C08947=1013.644,84.110,-119.825,166.038,58.565,160.621
C08948=1013.639,83.861,-119.809,166.035,58.575,160.623
C08949=1013.634,83.612,-119.793,166.034,58.586,160.624
C08950=1013.630,83.362,-119.778,166.031,58.596,160.626
C08951=1013.625,83.112,-119.762,166.029,58.606,160.627
C08952=1013.621,82.863,-119.746,166.027,58.617,160.629
C08953=1013.617,82.613,-119.730,166.025,58.627,160.630
C08954=1013.612,82.364,-119.715,166.022,58.638,160.632
C08955=1013.608,82.114,-119.699,166.021,58.647,160.633
C08956=1013.604,81.864,-119.683,166.018,58.658,160.634
C08957=1013.599,81.615,-119.668,166.016,58.669,160.636
C08958=1013.595,81.366,-119.652,166.014,58.678,160.637
C08959=1013.590,81.116,-119.636,166.011,58.689,160.639
C08960=1013.586,80.866,-119.621,166.009,58.699,160.640
C08961=1013.582,80.617,-119.605,166.007,58.709,160.642
C08962=1013.577,80.367,-119.589,166.004,58.719,160.643
C08963=1013.574,80.118,-119.574,166.002,58.730,160.644
C08964=1013.569,79.869,-119.558,166.000,58.740,160.646
C08965=1013.564,79.620,-119.543,165.997,58.750,160.647
C08966=1013.560,79.370,-119.527,165.996,58.760,160.649
C08967=1013.556,79.120,-119.511,165.994,58.771,160.650
C08968=1013.551,78.871,-119.495,165.992,58.781,160.652
C08969=1013.547,78.621,-119.480,165.989,58.791,160.653
C08970=1013.543,78.372,-119.464,165.986,58.801,160.654
C08971=1013.538,78.122,-119.448,165.984,58.811,160.656
C08972=1013.534,77.873,-119.432,165.982,58.822,160.657
C08973=1013.530,77.624,-119.417,165.981,58.832,160.659
C08974=1013.525,77.374,-119.402,165.978,58.842,160.660
C08975=1013.521,77.125,-119.386,165.976,58.852,160.662
C08976=1013.517,76.875,-119.370,165.973,58.862,160.663
C08977=1013.512,76.626,-119.354,165.972,58.872,160.664
C08978=1013.508,76.375,-119.339,165.969,58.882,160.666
C08979=1013.503,76.126,-119.324,165.968,58.893,160.668
C08980=1013.499,75.877,-119.308,165.965,58.903,160.669
C08981=1013.495,75.628,-119.293,165.963,58.913,160.670
C08982=1013.490,75.378,-119.278,165.960,58.923,160.672
C08983=1013.486,75.128,-119.263,165.958,58.933,160.673
C08984=1013.482,74.879,-119.247,165.956,58.943,160.674
C08985=1013.476,74.600,-119.230,165.953,58.955,160.676
C08986=1013.471,74.320,-119.213,165.951,58.966,160.678
C08987=1013.467,74.040,-119.196,165.949,58.977,160.679
C08988=1013.462,73.761,-119.178,165.946,58.988,160.681
C08989=1013.457,73.511,-119.164,165.944,58.998,160.682
C08990=1013.453,73.261,-119.148,165.942,59.008,160.683
C08991=1013.448,73.013,-119.133,165.940,59.018,160.685
C08992=1013.444,72.763,-119.118,165.938,59.029,160.687
C08993=1013.440,72.513,-119.102,165.936,59.039,160.688
C08994=1013.435,72.264,-119.087,165.933,59.049,160.689
C08995=1013.431,72.014,-119.072,165.932,59.059,160.691
C08996=1013.427,71.765,-119.057,165.929,59.069,160.692
C08997=1013.422,71.515,-119.041,165.927,59.079,160.694
C08998=1013.417,71.266,-119.026,165.925,59.089,160.695
C08999=1013.413,71.016,-119.011,165.922,59.098,160.696
C09000=1013.409,70.766,-118.995,165.921,59.108,160.698
C09001=1013.404,70.518,-118.981,165.918,59.119,160.699
C09002=1013.400,70.268,-118.966,165.916,59.128,160.700
C09003=1013.395,70.018,-118.950,165.914,59.139,160.702
C09004=1013.391,69.768,-118.935,165.912,59.148,160.703
C09005=1013.387,69.520,-118.921,165.910,59.158,160.705
C09006=1013.383,69.270,-118.905,165.908,59.169,160.706
C09007=1013.378,69.020,-118.890,165.906,59.178,160.708
C09008=1013.374,68.771,-118.875,165.904,59.188,160.709
C09009=1013.370,68.520,-118.860,165.901,59.198,160.710
C09010=1013.365,68.272,-118.845,165.899,59.208,160.712
C09011=1013.361,68.022,-118.829,165.898,59.217,160.713
C09012=1013.356,67.772,-118.814,165.895,59.228,160.714
C09013=1013.352,67.523,-118.799,165.893,59.237,160.716
C09014=1013.348,67.274,-118.785,165.892,59.247,160.717
C09015=1013.343,67.024,-118.769,165.888,59.257,160.718
C09016=1013.339,66.774,-118.754,165.887,59.267,160.720
C09017=1013.334,66.525,-118.739,165.885,59.277,160.721
C09018=1013.330,66.276,-118.725,165.883,59.287,160.723
C09019=1013.325,66.026,-118.709,165.881,59.297,160.724
C09020=1013.320,65.776,-118.695,165.879,59.306,160.725
C09021=1013.317,65.527,-118.679,165.876,59.316,160.727
C09022=1013.312,65.277,-118.665,165.874,59.326,160.728
C09023=1013.307,65.027,-118.651,165.873,59.336,160.730
C09024=1013.303,64.778,-118.635,165.871,59.345,160.731
C09025=1013.299,64.529,-118.621,165.868,59.355,160.732
C09026=1013.294,64.279,-118.606,165.866,59.365,160.734
C09027=1013.290,64.029,-118.590,165.864,59.374,160.735
C09028=1013.286,63.780,-118.576,165.863,59.384,160.737
C09029=1013.281,63.531,-118.561,165.860,59.394,160.738
C09030=1013.277,63.281,-118.546,165.858,59.403,160.739
C09031=1013.272,63.032,-118.531,165.856,59.413,160.741
C09032=1013.267,62.782,-118.517,165.855,59.423,160.742
C09033=1013.263,62.532,-118.502,165.851,59.433,160.743
C09034=1013.259,62.283,-118.487,165.850,59.442,160.745
C09035=1013.254,62.034,-118.473,165.848,59.452,160.746
C09036=1013.250,61.784,-118.458,165.846,59.461,160.747
C09037=1013.245,61.534,-118.444,165.843,59.472,160.749
C09038=1013.241,61.285,-118.430,165.842,59.482,160.750
C09039=1013.236,61.035,-118.414,165.840,59.491,160.751
C09040=1013.231,60.786,-118.400,165.838,59.501,160.753
C09041=1013.227,60.536,-118.386,165.835,59.511,160.754
C09042=1013.222,60.286,-118.371,165.833,59.520,160.756
C09043=1013.218,60.037,-118.357,165.832,59.530,160.757
C09044=1013.213,59.787,-118.343,165.829,59.539,160.758
C09045=1013.208,59.537,-118.328,165.827,59.549,160.760
C09046=1013.204,59.289,-118.314,165.825,59.559,160.761
C09047=1013.199,59.039,-118.299,165.823,59.568,160.762
C09048=1013.195,58.790,-118.285,165.822,59.578,160.764
C09049=1013.190,58.510,-118.269,165.819,59.589,160.765
C09050=1013.185,58.230,-118.253,165.817,59.600,160.767
C09051=1013.180,57.951,-118.236,165.814,59.610,160.768
C09052=1013.175,57.671,-118.220,165.813,59.621,160.770
C09053=1013.170,57.421,-118.205,165.810,59.630,160.771
C09054=1013.166,57.172,-118.191,165.809,59.640,160.773
C09055=1013.161,56.922,-118.177,165.807,59.649,160.774
C09056=1013.157,56.673,-118.163,165.803,59.659,160.775
C09057=1013.152,56.423,-118.148,165.802,59.669,160.776
C09058=1013.148,56.173,-118.134,165.800,59.678,160.778
C09059=1013.144,55.924,-118.120,165.798,59.688,160.779
C09060=1013.139,55.674,-118.105,165.796,59.697,160.780
C09061=1013.134,55.426,-118.090,165.794,59.706,160.782
C09062=1013.130,55.176,-118.076,165.792,59.715,160.783
C09063=1013.126,54.927,-118.062,165.790,59.725,160.784
C09064=1013.121,54.677,-118.047,165.788,59.734,160.786
C09065=1013.117,54.428,-118.033,165.786,59.743,160.787
C09066=1013.112,54.178,-118.019,165.785,59.753,160.788
C09067=1013.107,53.928,-118.004,165.782,59.762,160.790
C09068=1013.103,53.679,-117.990,165.780,59.772,160.791
C09069=1013.098,53.429,-117.976,165.778,59.781,160.792
C09070=1013.094,53.180,-117.962,165.776,59.790,160.793
C09071=1013.089,52.930,-117.947,165.775,59.800,160.795
C09072=1013.085,52.681,-117.933,165.773,59.809,160.796
C09073=1013.081,52.431,-117.919,165.771,59.818,160.797
C09074=1013.076,52.181,-117.905,165.769,59.827,160.799
C09075=1013.072,51.932,-117.890,165.767,59.836,160.800
C09076=1013.068,51.682,-117.876,165.765,59.845,160.801
C09077=1013.063,51.432,-117.862,165.763,59.854,160.802
C09078=1013.059,51.183,-117.848,165.761,59.864,160.804
C09079=1013.054,50.933,-117.833,165.759,59.873,160.805
C09080=1013.050,50.684,-117.819,165.758,59.881,160.806
C09081=1013.045,50.434,-117.805,165.755,59.891,160.807
C09082=1013.041,50.185,-117.791,165.753,59.900,160.809
C09083=1013.036,49.935,-117.776,165.751,59.909,160.810
C09084=1013.032,49.686,-117.762,165.749,59.918,160.811
C09085=1013.027,49.436,-117.747,165.748,59.927,160.813
C09086=1013.023,49.187,-117.733,165.746,59.936,160.814
C09087=1013.018,48.937,-117.719,165.744,59.945,160.815
C09088=1013.014,48.688,-117.705,165.742,59.954,160.816
C09089=1013.010,48.438,-117.690,165.741,59.963,160.818
C09090=1013.005,48.189,-117.676,165.739,59.972,160.819
C09091=1013.001,47.938,-117.663,165.736,59.981,160.820
C09092=1012.997,47.689,-117.648,165.734,59.990,160.821
C09093=1012.992,47.439,-117.634,165.733,59.999,160.823
C09094=1012.988,47.190,-117.620,165.731,60.008,160.824
C09095=1012.983,46.940,-117.605,165.729,60.017,160.825
C09096=1012.979,46.691,-117.591,165.727,60.025,160.826
C09097=1012.975,46.442,-117.577,165.725,60.034,160.827
C09098=1012.970,46.192,-117.563,165.723,60.043,160.829
C09099=1012.966,45.943,-117.549,165.721,60.051,160.830
C09100=1012.961,45.693,-117.534,165.719,60.061,160.831
C09101=1012.957,45.444,-117.520,165.718,60.069,160.832
C09102=1012.953,45.193,-117.506,165.715,60.078,160.833
C09103=1012.949,44.944,-117.492,165.713,60.087,160.835
C09104=1012.944,44.695,-117.478,165.712,60.096,160.836
C09105=1012.940,44.445,-117.464,165.709,60.104,160.837
C09106=1012.936,44.196,-117.450,165.708,60.113,160.838
C09107=1012.931,43.946,-117.435,165.706,60.121,160.839
C09108=1012.927,43.697,-117.421,165.705,60.130,160.841
C09109=1012.923,43.448,-117.407,165.703,60.139,160.842
C09110=1012.918,43.197,-117.393,165.701,60.147,160.843
C09111=1012.914,42.948,-117.379,165.699,60.157,160.844
C09112=1012.909,42.698,-117.365,165.697,60.165,160.845
C09113=1012.903,42.319,-117.343,165.694,60.177,160.847
C09114=1012.896,41.941,-117.322,165.691,60.191,160.849
C09115=1012.890,41.563,-117.301,165.688,60.204,160.851
C09116=1012.883,41.184,-117.280,165.685,60.217,160.852
C09117=1012.878,40.936,-117.266,165.684,60.225,160.854
C09118=1012.874,40.685,-117.253,165.681,60.234,160.855
C09119=1012.870,40.436,-117.239,165.680,60.243,160.856
C09120=1012.866,40.187,-117.225,165.678,60.251,160.857
C09121=1012.860,39.936,-117.211,165.677,60.260,160.859
C09122=1012.856,39.687,-117.197,165.674,60.268,160.859
C09123=1012.852,39.437,-117.184,165.673,60.277,160.861
C09124=1012.847,39.188,-117.170,165.670,60.286,160.862
C09125=1012.843,38.939,-117.156,165.669,60.294,160.863
C09126=1012.838,38.688,-117.142,165.668,60.302,160.864
C09127=1012.834,38.439,-117.128,165.665,60.311,160.865
C09128=1012.830,38.190,-117.115,165.663,60.319,160.866
C09129=1012.825,37.940,-117.101,165.661,60.328,160.868
C09130=1012.821,37.690,-117.087,165.660,60.336,160.869
C09131=1012.816,37.441,-117.074,165.658,60.344,160.870
C09132=1012.812,37.191,-117.060,165.656,60.353,160.871
C09133=1012.808,36.941,-117.046,165.655,60.361,160.872
C09134=1012.803,36.692,-117.033,165.653,60.369,160.873
C09135=1012.799,36.443,-117.019,165.650,60.378,160.874
C09136=1012.794,36.193,-117.005,165.649,60.386,160.875
C09137=1012.777,48.138,-118.086,165.708,60.195,160.855
C09138=1012.781,48.387,-118.101,165.711,60.187,160.854
C09139=1012.785,48.637,-118.115,165.711,60.178,160.853
C09140=1012.790,48.886,-118.129,165.714,60.169,160.851
C09141=1012.794,49.135,-118.143,165.715,60.161,160.850
C09142=1012.798,49.385,-118.158,165.717,60.152,160.849
C09143=1012.802,49.635,-118.171,165.720,60.143,160.848
C09144=1012.807,49.885,-118.185,165.721,60.134,160.847
C09145=1012.811,50.134,-118.200,165.723,60.125,160.845
C09146=1012.816,50.384,-118.214,165.725,60.116,160.844
C09147=1012.820,50.633,-118.228,165.727,60.108,160.843
C09148=1012.825,50.883,-118.243,165.729,60.099,160.842
C09149=1012.829,51.132,-118.257,165.730,60.090,160.840
C09150=1012.833,51.381,-118.271,165.732,60.081,160.839
C09151=1012.838,51.631,-118.285,165.735,60.072,160.838
C09152=1012.842,51.880,-118.299,165.737,60.063,160.837
C09153=1012.847,52.130,-118.314,165.738,60.055,160.836
C09154=1012.851,52.380,-118.328,165.740,60.045,160.834
C09155=1012.856,52.629,-118.342,165.742,60.036,160.833
C09156=1012.860,52.879,-118.356,165.743,60.027,160.832
C09157=1012.864,53.129,-118.370,165.745,60.018,160.830
C09158=1012.868,53.378,-118.384,165.748,60.010,160.829
C09159=1012.872,53.628,-118.399,165.750,60.001,160.828
C09160=1012.876,53.878,-118.413,165.752,59.991,160.827
C09161=1012.881,54.128,-118.428,165.753,59.983,160.826
C09162=1012.885,54.377,-118.442,165.755,59.974,160.824
C09163=1012.890,54.627,-118.456,165.757,59.964,160.823
C09164=1012.894,54.876,-118.470,165.759,59.955,160.822
C09165=1012.899,55.126,-118.485,165.761,59.946,160.821
C09166=1012.903,55.375,-118.499,165.763,59.937,160.819
C09167=1012.908,55.625,-118.514,165.764,59.927,160.818
C09168=1012.912,55.874,-118.528,165.766,59.918,160.816
C09169=1012.917,56.124,-118.542,165.768,59.909,160.815
C09170=1012.921,56.373,-118.556,165.770,59.900,160.814
C09171=1012.926,56.623,-118.571,165.772,59.891,160.813
C09172=1012.930,56.872,-118.585,165.774,59.881,160.811
C09173=1012.934,57.122,-118.599,165.776,59.872,160.810
C09174=1012.942,57.530,-118.623,165.779,59.857,160.808
C09175=1012.950,57.939,-118.647,165.783,59.842,160.806
C09176=1012.957,58.347,-118.669,165.785,59.826,160.803
C09177=1012.964,58.756,-118.693,165.789,59.811,160.802
C09178=1012.969,59.006,-118.708,165.791,59.801,160.800
C09179=1012.973,59.255,-118.722,165.793,59.792,160.799
C09180=1012.977,59.505,-118.736,165.795,59.783,160.798
C09181=1012.982,59.754,-118.750,165.796,59.773,160.796
C09182=1012.987,60.003,-118.765,165.799,59.764,160.795
C09183=1012.991,60.253,-118.780,165.801,59.755,160.794
C09184=1012.995,60.502,-118.794,165.802,59.745,160.792
C09185=1013.000,60.752,-118.808,165.804,59.736,160.791
C09186=1013.004,61.001,-118.822,165.806,59.726,160.789
C09187=1013.009,61.251,-118.837,165.808,59.716,160.788
C09188=1013.014,61.501,-118.851,165.811,59.706,160.787
C09189=1013.018,61.750,-118.865,165.813,59.697,160.785
C09190=1013.023,62.000,-118.880,165.814,59.687,160.784
C09191=1013.027,62.249,-118.894,165.816,59.678,160.783
C09192=1013.032,62.499,-118.909,165.818,59.668,160.781
C09193=1013.036,62.749,-118.924,165.820,59.659,160.780
C09194=1013.040,62.998,-118.938,165.822,59.650,160.779
C09195=1013.045,63.247,-118.954,165.824,59.640,160.777
C09196=1013.049,63.498,-118.969,165.826,59.631,160.776
C09197=1013.053,63.747,-118.983,165.828,59.620,160.775
C09198=1013.058,63.996,-118.998,165.831,59.611,160.773
C09199=1013.062,64.246,-119.013,165.832,59.601,160.772
C09200=1013.066,64.495,-119.027,165.834,59.592,160.771
C09201=1013.071,64.745,-119.042,165.836,59.582,160.769
C09202=1013.075,64.994,-119.057,165.838,59.573,160.768
C09203=1013.080,65.244,-119.071,165.840,59.563,160.766
C09204=1013.085,65.493,-119.086,165.843,59.554,160.765
C09205=1013.088,65.743,-119.101,165.844,59.544,160.764
C09206=1013.093,65.993,-119.116,165.847,59.535,160.763
C09207=1013.097,66.242,-119.131,165.848,59.525,160.761
C09208=1013.101,66.491,-119.145,165.850,59.515,160.759
C09209=1013.106,66.741,-119.161,165.853,59.505,160.758
C09210=1013.110,66.991,-119.176,165.854,59.496,160.757
C09211=1013.115,67.239,-119.191,165.857,59.486,160.756
C09212=1013.119,67.490,-119.206,165.858,59.477,160.754
C09213=1013.123,67.740,-119.220,165.860,59.467,160.753
C09214=1013.128,67.988,-119.235,165.863,59.457,160.752
C09215=1013.132,68.238,-119.250,165.865,59.447,160.750
C09216=1013.136,68.488,-119.266,165.866,59.437,160.749
C09217=1013.141,68.738,-119.280,165.868,59.428,160.747
C09218=1013.145,68.987,-119.296,165.871,59.418,160.746
C09219=1013.149,69.237,-119.310,165.873,59.408,160.745
C09220=1013.154,69.486,-119.326,165.875,59.399,160.743
C09221=1013.158,69.735,-119.341,165.876,59.389,160.742
C09222=1013.162,69.985,-119.356,165.879,59.379,160.740
C09223=1013.167,70.234,-119.371,165.881,59.369,160.739
C09224=1013.171,70.484,-119.386,165.883,59.360,160.738
C09225=1013.176,70.733,-119.401,165.885,59.350,160.736
C09226=1013.180,70.983,-119.416,165.887,59.340,160.735
C09227=1013.184,71.233,-119.431,165.889,59.330,160.733
C09228=1013.189,71.482,-119.447,165.892,59.320,160.732
C09229=1013.192,71.731,-119.461,165.894,59.311,160.731
C09230=1013.197,71.981,-119.477,165.895,59.301,160.729
C09231=1013.202,72.230,-119.492,165.898,59.290,160.728
C09232=1013.205,72.480,-119.507,165.899,59.281,160.727
C09233=1013.210,72.729,-119.522,165.901,59.271,160.725
C09234=1013.214,72.979,-119.537,165.904,59.261,160.724
C09235=1013.219,73.229,-119.552,165.905,59.251,160.722
C09236=1013.223,73.478,-119.568,165.909,59.241,160.721
C09237=1013.228,73.727,-119.582,165.910,59.231,160.720
C09238=1013.232,74.006,-119.600,165.912,59.220,160.718
C09239=1013.237,74.286,-119.617,165.915,59.209,160.717
C09240=1013.242,74.566,-119.634,165.917,59.197,160.715
C09241=1013.248,74.845,-119.651,165.919,59.186,160.713
C09242=1013.251,75.095,-119.666,165.921,59.176,160.712
C09243=1013.255,75.344,-119.682,165.923,59.166,160.710
C09244=1013.261,75.594,-119.697,165.926,59.156,160.709
C09245=1013.265,75.843,-119.712,165.927,59.146,160.707
C09246=1013.269,76.093,-119.728,165.930,59.136,160.706
C09247=1013.273,76.342,-119.742,165.932,59.126,160.705
C09248=1013.278,76.591,-119.758,165.935,59.116,160.703
C09249=1013.282,76.841,-119.774,165.936,59.106,160.702
C09250=1013.286,77.091,-119.789,165.939,59.095,160.700
C09251=1013.291,77.341,-119.804,165.941,59.086,160.699
C09252=1013.295,77.590,-119.820,165.942,59.076,160.697
C09253=1013.299,77.839,-119.835,165.945,59.066,160.696
C09254=1013.303,78.089,-119.851,165.947,59.056,160.695
C09255=1013.308,78.338,-119.867,165.949,59.046,160.693
C09256=1013.312,78.588,-119.883,165.951,59.036,160.692
C09257=1013.316,78.837,-119.898,165.954,59.025,160.691
C09258=1013.320,79.087,-119.914,165.955,59.016,160.689
C09259=1013.324,79.336,-119.929,165.958,59.005,160.688
C09260=1013.329,79.586,-119.944,165.960,58.996,160.686
C09261=1013.333,79.835,-119.960,165.963,58.985,160.685
C09262=1013.338,80.085,-119.976,165.964,58.976,160.683
C09263=1013.342,80.334,-119.991,165.966,58.965,160.682
C09264=1013.346,80.584,-120.007,165.969,58.954,160.681
C09265=1013.350,80.834,-120.023,165.971,58.945,160.679
C09266=1013.354,81.082,-120.038,165.974,58.934,160.678
C09267=1013.358,81.332,-120.054,165.975,58.925,160.676
C09268=1013.363,81.581,-120.069,165.977,58.914,160.675
C09269=1013.368,81.831,-120.085,165.979,58.904,160.673
C09270=1013.372,82.080,-120.101,165.982,58.894,160.672
C09271=1013.376,82.330,-120.116,165.985,58.883,160.671
C09272=1013.381,82.580,-120.132,165.986,58.873,160.669
C09273=1013.385,82.829,-120.148,165.988,58.863,160.667
C09274=1013.389,83.078,-120.163,165.991,58.852,160.666
C09275=1013.393,83.328,-120.179,165.992,58.842,160.664
C09276=1013.398,83.577,-120.194,165.995,58.832,160.663
C09277=1013.402,83.826,-120.210,165.998,58.821,160.662
C09278=1013.407,84.076,-120.226,165.999,58.811,160.660
C09279=1013.411,84.326,-120.242,166.002,58.801,160.659
C09280=1013.415,84.575,-120.257,166.005,58.790,160.657
C09281=1013.420,84.825,-120.273,166.006,58.780,160.656
C09282=1013.424,85.074,-120.289,166.008,58.770,160.654
C09283=1013.428,85.324,-120.305,166.011,58.760,160.653
C09284=1013.433,85.573,-120.320,166.013,58.749,160.652
C09285=1013.438,85.823,-120.336,166.015,58.739,160.650
C09286=1013.441,86.072,-120.351,166.017,58.728,160.648
C09287=1013.446,86.321,-120.367,166.020,58.718,160.647
C09288=1013.450,86.571,-120.383,166.022,58.707,160.646
C09289=1013.454,86.820,-120.398,166.024,58.697,160.644
C09290=1013.458,87.070,-120.414,166.026,58.686,160.642
C09291=1013.463,87.319,-120.430,166.029,58.676,160.641
C09292=1013.467,87.568,-120.446,166.031,58.665,160.640
C09293=1013.472,87.818,-120.462,166.034,58.655,160.638
C09294=1013.477,88.067,-120.477,166.035,58.644,160.637
C09295=1013.481,88.317,-120.493,166.038,58.633,160.635
C09296=1013.485,88.566,-120.509,166.040,58.623,160.634
C09297=1013.490,88.816,-120.525,166.043,58.612,160.632
C09298=1013.493,89.066,-120.541,166.045,58.602,160.631
C09299=1013.498,89.315,-120.558,166.047,58.592,160.629
C09300=1013.502,89.564,-120.573,166.049,58.581,160.628
C09301=1013.506,89.814,-120.589,166.052,58.571,160.627
C09302=1013.511,90.094,-120.608,166.055,58.559,160.625
C09303=1013.516,90.373,-120.625,166.057,58.547,160.623
C09304=1013.521,90.653,-120.644,166.060,58.536,160.622
C09305=1013.526,90.932,-120.662,166.063,58.524,160.620
C09306=1013.530,91.182,-120.677,166.065,58.513,160.618
C09307=1013.534,91.431,-120.694,166.067,58.503,160.617
C09308=1013.538,91.681,-120.710,166.069,58.492,160.615
C09309=1013.542,91.930,-120.726,166.072,58.482,160.614
C09310=1013.547,92.179,-120.742,166.074,58.471,160.612
C09311=1013.551,92.429,-120.758,166.077,58.461,160.611
C09312=1013.555,92.679,-120.775,166.079,58.450,160.610
C09313=1013.560,92.928,-120.791,166.080,58.440,160.608
C09314=1013.564,93.177,-120.807,166.083,58.430,160.607
C09315=1013.568,93.426,-120.823,166.085,58.419,160.605
C09316=1013.573,93.676,-120.839,166.088,58.408,160.603
C09317=1013.576,93.926,-120.855,166.091,58.398,160.602
C09318=1013.581,94.175,-120.872,166.093,58.387,160.601
C09319=1013.586,94.425,-120.888,166.095,58.376,160.599
C09320=1013.590,94.675,-120.904,166.098,58.366,160.598
C09321=1013.595,94.923,-120.920,166.100,58.355,160.596
C09322=1013.598,95.173,-120.937,166.103,58.344,160.595
C09323=1013.603,95.422,-120.953,166.104,58.334,160.593
C09324=1013.607,95.672,-120.969,166.107,58.323,160.592
C09325=1013.612,95.921,-120.985,166.109,58.313,160.590
C09326=1013.616,96.170,-121.001,166.111,58.302,160.589
C09327=1013.620,96.420,-121.017,166.114,58.291,160.587
C09328=1013.624,96.669,-121.034,166.116,58.280,160.585
C09329=1013.629,96.919,-121.050,166.119,58.270,160.584
C09330=1013.633,97.168,-121.066,166.121,58.259,160.583
C09331=1013.637,97.418,-121.083,166.124,58.248,160.581
C09332=1013.642,97.667,-121.099,166.126,58.237,160.579
C09333=1013.646,97.917,-121.115,166.128,58.226,160.578
C09334=1013.651,98.166,-121.132,166.131,58.215,160.576
C09335=1013.655,98.415,-121.147,166.133,58.205,160.575
C09336=1013.659,98.665,-121.165,166.135,58.194,160.573
C09337=1013.663,98.914,-121.180,166.138,58.184,160.572
C09338=1013.667,99.164,-121.197,166.141,58.173,160.570
C09339=1013.672,99.413,-121.213,166.143,58.162,160.569
C09340=1013.676,99.663,-121.231,166.145,58.151,160.567
C09341=1013.681,99.912,-121.247,166.148,58.141,160.566
C09342=1013.684,100.162,-121.263,166.151,58.130,160.565
C09343=1013.689,100.411,-121.280,166.153,58.119,160.563
C09344=1013.693,100.660,-121.297,166.155,58.108,160.561
C09345=1013.697,100.909,-121.314,166.158,58.098,160.560
C09346=1013.701,101.159,-121.330,166.160,58.087,160.558
C09347=1013.706,101.409,-121.347,166.163,58.077,160.557
C09348=1013.710,101.658,-121.364,166.165,58.066,160.556
C09349=1013.714,101.908,-121.380,166.168,58.055,160.554
C09350=1013.718,102.157,-121.397,166.170,58.044,160.553
C09351=1013.723,102.406,-121.413,166.172,58.033,160.551
C09352=1013.726,102.656,-121.430,166.175,58.022,160.549
C09353=1013.732,102.905,-121.446,166.177,58.012,160.548
C09354=1013.735,103.155,-121.463,166.181,58.000,160.547
C09355=1013.740,103.404,-121.480,166.183,57.989,160.545
C09356=1013.744,103.653,-121.496,166.186,57.979,160.544
C09357=1013.748,103.902,-121.513,166.188,57.968,160.542
C09358=1013.753,104.152,-121.530,166.190,57.957,160.540
C09359=1013.757,104.401,-121.547,166.193,57.946,160.539
C09360=1013.761,104.651,-121.563,166.195,57.935,160.537
C09361=1013.766,104.900,-121.580,166.198,57.925,160.536
C09362=1013.769,105.149,-121.597,166.200,57.914,160.534
C09363=1013.775,105.399,-121.613,166.202,57.903,160.533
C09364=1013.778,105.648,-121.631,166.206,57.892,160.531
C09365=1013.783,105.898,-121.646,166.208,57.881,160.530
C09366=1013.788,106.177,-121.666,166.211,57.869,160.528
C09367=1013.793,106.458,-121.684,166.214,57.857,160.527
C09368=1013.797,106.738,-121.703,166.216,57.844,160.525
C09369=1013.802,107.018,-121.721,166.219,57.832,160.523
C09370=1013.806,107.268,-121.739,166.223,57.821,160.522
C09371=1013.811,107.517,-121.755,166.225,57.810,160.520
C09372=1013.815,107.766,-121.772,166.228,57.799,160.519
C09373=1013.820,108.015,-121.789,166.229,57.788,160.517
C09374=1013.824,108.265,-121.806,166.233,57.777,160.516
C09375=1013.828,108.514,-121.822,166.235,57.766,160.514
C09376=1013.832,108.764,-121.839,166.238,57.755,160.512
C09377=1013.836,109.013,-121.856,166.240,57.744,160.511
C09378=1013.841,109.263,-121.873,166.243,57.733,160.509
C09379=1013.845,109.512,-121.890,166.246,57.722,160.508
C09380=1013.849,109.761,-121.907,166.249,57.711,160.507
C09381=1013.854,110.011,-121.924,166.251,57.700,160.505
C09382=1013.858,110.260,-121.941,166.253,57.689,160.503
C09383=1013.862,110.509,-121.958,166.256,57.678,160.502
C09384=1013.867,110.758,-121.975,166.259,57.667,160.500
C09385=1013.871,111.008,-121.992,166.262,57.656,160.499
C09386=1013.875,111.258,-122.009,166.264,57.646,160.497
C09387=1013.879,111.507,-122.026,166.266,57.634,160.496
C09388=1013.884,111.756,-122.043,166.270,57.623,160.494
C09389=1013.888,112.006,-122.060,166.272,57.612,160.493
C09390=1013.892,112.255,-122.077,166.275,57.601,160.491
C09391=1013.897,112.504,-122.096,166.277,57.591,160.490
C09392=1013.900,112.754,-122.113,166.280,57.580,160.488
C09393=1013.904,113.003,-122.130,166.282,57.569,160.487
C09394=1013.909,113.253,-122.147,166.285,57.558,160.485
C09395=1013.913,113.502,-122.165,166.288,57.547,160.484
C09396=1013.917,113.751,-122.182,166.291,57.536,160.482
C09397=1013.921,114.001,-122.199,166.293,57.526,160.481
C09398=1013.925,114.250,-122.217,166.295,57.514,160.479
C09399=1013.929,114.499,-122.234,166.298,57.503,160.478
C09400=1013.934,114.749,-122.252,166.301,57.492,160.476
C09401=1013.938,114.998,-122.269,166.304,57.482,160.475
C09402=1013.942,115.247,-122.286,166.306,57.471,160.473
C09403=1013.946,115.497,-122.304,166.309,57.460,160.472
C09404=1013.950,115.746,-122.321,166.313,57.449,160.470
C09405=1013.954,115.995,-122.338,166.315,57.437,160.469
C09406=1013.959,116.245,-122.356,166.317,57.427,160.467
C09407=1013.963,116.494,-122.374,166.320,57.416,160.466
C09408=1013.967,116.744,-122.391,166.323,57.405,160.464
C09409=1013.971,116.993,-122.408,166.326,57.394,160.463
C09410=1013.975,117.242,-122.426,166.328,57.383,160.461
C09411=1013.980,117.492,-122.443,166.330,57.372,160.460
C09412=1013.984,117.741,-122.460,166.334,57.361,160.458
C09413=1013.988,117.990,-122.479,166.337,57.350,160.457
C09414=1013.992,118.239,-122.496,166.339,57.339,160.455
C09415=1013.996,118.489,-122.513,166.342,57.327,160.454
C09416=1014.001,118.738,-122.531,166.345,57.317,160.452
C09417=1014.005,118.987,-122.548,166.347,57.305,160.450
C09418=1014.009,119.237,-122.565,166.350,57.294,160.449
C09419=1014.013,119.486,-122.584,166.353,57.283,160.448
C09420=1014.017,119.736,-122.601,166.355,57.272,160.446
C09421=1014.021,119.986,-122.618,166.359,57.261,160.445
C09422=1014.025,120.234,-122.636,166.361,57.250,160.443
C09423=1014.030,120.484,-122.654,166.363,57.239,160.441
C09424=1014.034,120.733,-122.671,166.367,57.227,160.440
C09425=1014.038,120.983,-122.689,166.370,57.217,160.439
C09426=1014.042,121.232,-122.706,166.373,57.205,160.437
C09427=1014.047,121.481,-122.724,166.375,57.194,160.435
C09428=1014.051,121.731,-122.741,166.378,57.184,160.434
C09429=1014.055,121.981,-122.759,166.381,57.172,160.432
C09430=1014.060,122.260,-122.778,166.383,57.159,160.431
C09431=1014.065,122.541,-122.798,166.388,57.147,160.429
C09432=1014.070,122.820,-122.818,166.390,57.134,160.427
C09433=1014.075,123.101,-122.838,166.394,57.121,160.426
C09434=1014.079,123.350,-122.855,166.396,57.111,160.424
C09435=1014.084,123.599,-122.873,166.399,57.099,160.422
C09436=1014.088,123.848,-122.890,166.402,57.088,160.421
C09437=1014.093,124.098,-122.908,166.405,57.076,160.419
C09438=1014.096,124.347,-122.925,166.408,57.066,160.418
C09439=1014.101,124.596,-122.943,166.411,57.054,160.416
C09440=1014.105,124.846,-122.960,166.414,57.043,160.415
C09441=1014.110,125.095,-122.979,166.416,57.032,160.413
C09442=1014.114,125.344,-122.996,166.419,57.021,160.412
C09443=1014.119,125.594,-123.014,166.423,57.009,160.410
C09444=1014.122,125.843,-123.031,166.425,56.998,160.409
C09445=1014.127,126.092,-123.049,166.428,56.986,160.407
C09446=1014.131,126.342,-123.066,166.431,56.976,160.406
C09447=1014.136,126.591,-123.084,166.434,56.964,160.404
C09448=1014.140,126.840,-123.101,166.437,56.953,160.403
C09449=1014.144,127.089,-123.120,166.440,56.941,160.401
C09450=1014.148,127.340,-123.138,166.442,56.930,160.399
C09451=1014.152,127.588,-123.155,166.446,56.919,160.398
C09452=1014.157,127.838,-123.173,166.448,56.907,160.396
C09453=1014.161,128.087,-123.191,166.452,56.896,160.395
C09454=1014.166,128.337,-123.208,166.455,56.885,160.394
C09455=1014.170,128.586,-123.226,166.457,56.873,160.392
C09456=1014.174,128.835,-123.244,166.461,56.862,160.390
C09457=1014.179,129.085,-123.262,166.463,56.851,160.389
C09458=1014.183,129.334,-123.279,166.466,56.839,160.387
C09459=1014.188,129.583,-123.297,166.469,56.828,160.386
C09460=1014.192,129.833,-123.316,166.472,56.817,160.384
C09461=1014.196,130.082,-123.333,166.475,56.806,160.383
C09462=1014.201,130.331,-123.351,166.478,56.794,160.381
C09463=1014.204,130.580,-123.370,166.481,56.784,160.380
C09464=1014.209,130.830,-123.387,166.485,56.772,160.378
C09465=1014.213,131.080,-123.405,166.487,56.761,160.377
C09466=1014.217,131.329,-123.424,166.490,56.749,160.375
C09467=1014.222,131.578,-123.442,166.493,56.739,160.374
C09468=1014.226,131.828,-123.461,166.496,56.727,160.372
C09469=1014.230,132.076,-123.479,166.500,56.716,160.371
C09470=1014.234,132.326,-123.496,166.502,56.705,160.369
C09471=1014.238,132.575,-123.514,166.506,56.694,160.368
C09472=1014.242,132.824,-123.533,166.508,56.682,160.366
C09473=1014.246,133.074,-123.551,166.512,56.671,160.365
C09474=1014.251,133.323,-123.569,166.514,56.660,160.363
C09475=1014.255,133.572,-123.587,166.517,56.648,160.362
C09476=1014.259,133.822,-123.606,166.521,56.637,160.360
C09477=1014.264,134.070,-123.624,166.523,56.626,160.359
C09478=1014.268,134.320,-123.642,166.527,56.615,160.357
C09479=1014.272,134.570,-123.660,166.529,56.603,160.356
C09480=1014.276,134.819,-123.678,166.533,56.592,160.354
C09481=1014.280,135.068,-123.697,166.536,56.581,160.353
C09482=1014.285,135.318,-123.715,166.539,56.569,160.351
C09483=1014.289,135.567,-123.734,166.542,56.558,160.350
C09484=1014.293,135.816,-123.751,166.545,56.547,160.348
C09485=1014.298,136.065,-123.769,166.548,56.535,160.346
C09486=1014.302,136.315,-123.788,166.552,56.524,160.345
C09487=1014.306,136.564,-123.806,166.554,56.513,160.343
C09488=1014.310,136.813,-123.825,166.558,56.502,160.342
C09489=1014.315,137.063,-123.843,166.560,56.491,160.340
C09490=1014.319,137.312,-123.862,166.563,56.479,160.339
C09491=1014.323,137.561,-123.879,166.567,56.468,160.338
C09492=1014.327,137.811,-123.898,166.570,56.457,160.336
C09493=1014.332,138.060,-123.917,166.573,56.445,160.334
C09494=1014.337,138.340,-123.938,166.577,56.433,160.333
C09495=1014.341,138.619,-123.959,166.580,56.420,160.331
C09496=1014.345,138.900,-123.979,166.584,56.407,160.330
C09497=1014.351,139.180,-124.000,166.588,56.395,160.328
C09498=1014.355,139.430,-124.019,166.590,56.383,160.326
C09499=1014.360,139.679,-124.037,166.594,56.372,160.325
C09500=1014.363,139.928,-124.056,166.596,56.361,160.323
C09501=1014.367,140.177,-124.075,166.599,56.349,160.322
C09502=1014.372,140.426,-124.093,166.603,56.338,160.320
C09503=1014.376,140.676,-124.112,166.606,56.327,160.319
C09504=1014.380,140.926,-124.131,166.609,56.316,160.317
C09505=1014.384,141.174,-124.149,166.613,56.304,160.316
C09506=1014.389,141.423,-124.168,166.615,56.293,160.314
C09507=1014.393,141.673,-124.187,166.619,56.282,160.313
C09508=1014.398,141.922,-124.205,166.622,56.271,160.311
C09509=1014.402,142.172,-124.224,166.625,56.259,160.310
C09510=1014.405,142.420,-124.243,166.628,56.248,160.308
C09511=1014.410,142.670,-124.261,166.632,56.237,160.307
C09512=1014.414,142.919,-124.280,166.634,56.225,160.305
C09513=1014.418,143.169,-124.299,166.638,56.214,160.304
C09514=1014.423,143.418,-124.317,166.642,56.203,160.302
C09515=1014.427,143.667,-124.336,166.645,56.191,160.301
C09516=1014.431,143.916,-124.355,166.647,56.180,160.299
C09517=1014.436,144.166,-124.373,166.651,56.169,160.298
C09518=1014.440,144.415,-124.392,166.655,56.157,160.296
C09519=1014.445,144.664,-124.410,166.658,56.146,160.295
C09520=1014.449,144.914,-124.429,166.660,56.134,160.293
C09521=1014.453,145.163,-124.449,166.664,56.123,160.292
C09522=1014.456,145.412,-124.467,166.668,56.112,160.291
C09523=1014.462,145.661,-124.486,166.671,56.100,160.289
C09524=1014.466,145.910,-124.505,166.674,56.090,160.288
C09525=1014.470,146.160,-124.523,166.678,56.078,160.286
C09526=1014.474,146.409,-124.543,166.681,56.066,160.285
C09527=1014.478,146.659,-124.562,166.683,56.055,160.283
C09528=1014.482,146.908,-124.581,166.687,56.044,160.282
C09529=1014.486,147.157,-124.600,166.691,56.033,160.280
C09530=1014.492,147.406,-124.619,166.694,56.021,160.279
C09531=1014.495,147.655,-124.637,166.697,56.010,160.277
C09532=1014.499,147.904,-124.657,166.701,55.999,160.276
C09533=1014.503,148.154,-124.675,166.704,55.987,160.274
C09534=1014.508,148.403,-124.695,166.708,55.976,160.273
C09535=1014.512,148.652,-124.714,166.710,55.965,160.271
C09536=1014.516,148.901,-124.733,166.714,55.953,160.270
C09537=1014.520,149.151,-124.753,166.718,55.943,160.268
C09538=1014.524,149.400,-124.771,166.721,55.931,160.267
C09539=1014.529,149.649,-124.791,166.724,55.920,160.265
C09540=1014.533,149.899,-124.810,166.727,55.908,160.264
C09541=1014.537,150.148,-124.829,166.731,55.897,160.262
C09542=1014.542,150.397,-124.848,166.735,55.886,160.261
C09543=1014.546,150.646,-124.867,166.737,55.874,160.259
C09544=1014.551,150.895,-124.886,166.741,55.864,160.258
C09545=1014.554,151.144,-124.904,166.745,55.852,160.257
C09546=1014.558,151.393,-124.924,166.748,55.840,160.255
C09547=1014.563,151.642,-124.943,166.752,55.829,160.254
C09548=1014.567,151.892,-124.962,166.754,55.818,160.252
C09549=1014.571,152.141,-124.982,166.758,55.807,160.251
C09550=1014.576,152.390,-125.001,166.762,55.795,160.249
C09551=1014.580,152.640,-125.020,166.765,55.784,160.248
C09552=1014.584,152.889,-125.039,166.769,55.773,160.246
C09553=1014.588,153.138,-125.059,166.771,55.761,160.245
C09554=1014.593,153.387,-125.078,166.775,55.750,160.243
C09555=1014.597,153.637,-125.097,166.779,55.738,160.242
C09556=1014.600,153.886,-125.117,166.783,55.727,160.240
C09557=1014.605,154.135,-125.137,166.786,55.716,160.239
C09558=1014.610,154.416,-125.159,166.790,55.703,160.237
C09559=1014.615,154.695,-125.180,166.793,55.691,160.236
C09560=1014.620,154.975,-125.202,166.797,55.678,160.234
C09561=1014.624,155.255,-125.223,166.801,55.666,160.232
C09562=1014.629,155.505,-125.243,166.805,55.654,160.231
C09563=1014.633,155.754,-125.263,166.808,55.642,160.229
C09564=1014.637,156.004,-125.283,166.812,55.631,160.228
C09565=1014.641,156.253,-125.302,166.816,55.620,160.227
C09566=1014.645,156.502,-125.321,166.819,55.608,160.225
C09567=1014.650,156.751,-125.340,166.823,55.597,160.224
C09568=1014.654,157.000,-125.360,166.826,55.586,160.222
C09569=1014.658,157.249,-125.379,166.829,55.574,160.220
C09570=1014.663,157.499,-125.399,166.833,55.563,160.219
C09571=1014.667,157.748,-125.418,166.837,55.552,160.218
C09572=1014.672,157.997,-125.438,166.840,55.540,160.216
C09573=1014.676,158.246,-125.457,166.844,55.529,160.215
C09574=1014.680,158.496,-125.478,166.848,55.518,160.214
C09575=1014.684,158.745,-125.498,166.850,55.507,160.212
C09576=1014.688,158.994,-125.517,166.854,55.495,160.210
C09577=1014.692,159.243,-125.537,166.858,55.484,160.209
C09578=1014.696,159.492,-125.557,166.862,55.473,160.208
C09579=1014.700,159.742,-125.577,166.865,55.463,160.206
C09580=1014.704,159.991,-125.598,166.868,55.451,160.205
C09581=1014.708,160.240,-125.617,166.873,55.440,160.204
C09582=1014.712,160.490,-125.638,166.876,55.429,160.202
C09583=1014.716,160.739,-125.657,166.880,55.417,160.201
C09584=1014.720,160.987,-125.678,166.883,55.407,160.199
C09585=1014.725,161.236,-125.697,166.886,55.395,160.198
C09586=1014.728,161.486,-125.717,166.891,55.384,160.197
C09587=1014.732,161.735,-125.737,166.894,55.373,160.195
C09588=1014.737,161.984,-125.758,166.898,55.361,160.194
C09589=1014.741,162.234,-125.778,166.901,55.351,160.192
C09590=1014.745,162.483,-125.798,166.905,55.340,160.191
C09591=1014.749,162.732,-125.818,166.908,55.328,160.189
C09592=1014.753,162.980,-125.838,166.912,55.317,160.188
C09593=1014.757,163.230,-125.858,166.916,55.306,160.186
C09594=1014.761,163.479,-125.878,166.920,55.294,160.185
C09595=1014.766,163.728,-125.898,166.923,55.284,160.184
C09596=1014.769,163.978,-125.919,166.926,55.272,160.182
C09597=1014.774,164.227,-125.938,166.930,55.261,160.181
C09598=1014.778,164.475,-125.959,166.934,55.250,160.179
C09599=1014.781,164.725,-125.979,166.938,55.239,160.178
C09600=1014.786,164.975,-125.999,166.941,55.227,160.176
C09601=1014.790,165.223,-126.019,166.946,55.216,160.175
C09602=1014.795,165.472,-126.039,166.949,55.205,160.174
C09603=1014.798,165.721,-126.060,166.952,55.194,160.172
C09604=1014.803,165.971,-126.080,166.956,55.183,160.171
C09605=1014.807,166.220,-126.100,166.960,55.172,160.169
C09606=1014.811,166.469,-126.120,166.963,55.160,160.168
C09607=1014.815,166.718,-126.140,166.968,55.150,160.167
C09608=1014.820,166.967,-126.161,166.971,55.138,160.165
C09609=1014.824,167.216,-126.180,166.975,55.127,160.164
C09610=1014.828,167.466,-126.201,166.979,55.115,160.162
C09611=1014.832,167.714,-126.221,166.983,55.104,160.161
C09612=1014.837,167.964,-126.241,166.987,55.093,160.160
C09613=1014.841,168.213,-126.262,166.990,55.082,160.158
C09614=1014.845,168.462,-126.281,166.995,55.071,160.157
C09615=1014.849,168.711,-126.303,166.998,55.059,160.155
C09616=1014.854,168.960,-126.322,167.002,55.048,160.154
C09617=1014.858,169.209,-126.343,167.006,55.036,160.153
C09618=1014.862,169.459,-126.363,167.010,55.026,160.151
C09619=1014.867,169.708,-126.383,167.014,55.014,160.150
C09620=1014.870,169.957,-126.404,167.017,55.003,160.148
C09621=1014.875,170.206,-126.424,167.021,54.991,160.147
C09622=1014.879,170.486,-126.447,167.025,54.979,160.145
C09623=1014.884,170.766,-126.469,167.030,54.966,160.144
C09624=1014.889,171.046,-126.492,167.034,54.954,160.142
C09625=1014.894,171.325,-126.515,167.038,54.941,160.141
C09626=1014.898,171.575,-126.536,167.042,54.930,160.139
C09627=1014.903,171.824,-126.556,167.045,54.918,160.138
C09628=1014.906,172.073,-126.576,167.051,54.907,160.137
C09629=1014.912,172.322,-126.597,167.055,54.896,160.135
C09630=1014.916,172.571,-126.618,167.058,54.885,160.134
C09631=1014.921,172.821,-126.637,167.062,54.873,160.132
C09632=1014.924,173.069,-126.658,167.066,54.862,160.131
C09633=1014.928,173.319,-126.678,167.070,54.851,160.130
C09634=1014.933,173.568,-126.699,167.074,54.840,160.128
C09635=1014.937,173.816,-126.720,167.078,54.828,160.127
C09636=1014.942,174.066,-126.739,167.081,54.817,160.125
C09637=1014.946,174.315,-126.760,167.085,54.805,160.124
C09638=1014.951,174.564,-126.781,167.089,54.795,160.122
C09639=1014.955,174.813,-126.801,167.094,54.783,160.121
C09640=1014.959,175.062,-126.822,167.098,54.772,160.120
C09641=1014.964,175.311,-126.842,167.102,54.760,160.118
C09642=1014.968,175.561,-126.862,167.106,54.749,160.117
C09643=1014.972,175.810,-126.883,167.109,54.737,160.115
C09644=1014.977,176.058,-126.904,167.114,54.727,160.114
C09645=1014.981,176.308,-126.925,167.117,54.715,160.113
C09646=1014.986,176.557,-126.944,167.122,54.704,160.111
C09647=1014.990,176.806,-126.965,167.126,54.692,160.110
C09648=1014.994,177.055,-126.986,167.130,54.681,160.108
C09649=1014.999,177.304,-127.007,167.134,54.670,160.107
C09650=1015.003,177.554,-127.027,167.137,54.658,160.105
C09651=1015.008,177.803,-127.047,167.142,54.648,160.104
C09652=1015.012,178.051,-127.068,167.147,54.636,160.103
C09653=1015.017,178.301,-127.089,167.150,54.624,160.102
C09654=1015.021,178.549,-127.109,167.154,54.613,160.100
C09655=1015.026,178.799,-127.130,167.158,54.602,160.099
C09656=1015.031,179.049,-127.150,167.162,54.590,160.097
C09657=1015.035,179.297,-127.171,167.167,54.579,160.096
C09658=1015.039,179.547,-127.192,167.171,54.568,160.095
C09659=1015.044,179.795,-127.212,167.175,54.557,160.093
C09660=1015.048,180.045,-127.234,167.179,54.545,160.092
C09661=1015.052,180.294,-127.254,167.184,54.534,160.090
C09662=1015.057,180.543,-127.274,167.188,54.522,160.089
C09663=1015.062,180.792,-127.295,167.191,54.511,160.087
C09664=1015.067,181.041,-127.316,167.195,54.500,160.086
C09665=1015.071,181.290,-127.337,167.200,54.488,160.085
C09666=1015.075,181.539,-127.358,167.204,54.477,160.084
C09667=1015.079,181.788,-127.379,167.208,54.466,160.082
C09668=1015.084,182.038,-127.400,167.212,54.455,160.081
C09669=1015.089,182.287,-127.421,167.217,54.444,160.079
C09670=1015.092,182.536,-127.443,167.220,54.433,160.078
C09671=1015.097,182.785,-127.464,167.225,54.422,160.077
C09672=1015.100,183.034,-127.485,167.229,54.411,160.075
C09673=1015.105,183.283,-127.507,167.233,54.400,160.074
C09674=1015.108,183.532,-127.528,167.238,54.389,160.073
C09675=1015.113,183.781,-127.549,167.242,54.377,160.071
C09676=1015.117,184.031,-127.571,167.246,54.367,160.070
C09677=1015.122,184.279,-127.592,167.250,54.355,160.069
C09678=1015.125,184.529,-127.614,167.255,54.345,160.068
C09679=1015.130,184.777,-127.636,167.258,54.333,160.066
C09680=1015.134,185.026,-127.656,167.262,54.322,160.065
C09681=1015.138,185.276,-127.678,167.267,54.312,160.063
C09682=1015.143,185.525,-127.700,167.271,54.300,160.062
C09683=1015.147,185.773,-127.721,167.276,54.289,160.061
C09684=1015.151,186.023,-127.742,167.280,54.278,160.059
C09685=1015.155,186.272,-127.764,167.284,54.267,160.058
C09686=1015.160,186.551,-127.788,167.289,54.255,160.057
C09687=1015.165,186.831,-127.812,167.293,54.243,160.055
C09688=1015.170,187.110,-127.837,167.299,54.230,160.054
C09689=1015.175,187.390,-127.861,167.303,54.218,160.052
C09690=1015.179,187.639,-127.881,167.307,54.206,160.051
C09691=1015.183,187.888,-127.904,167.312,54.196,160.050
C09692=1015.187,188.138,-127.925,167.317,54.184,160.048
C09693=1015.192,188.387,-127.947,167.320,54.173,160.047
C09694=1015.196,188.635,-127.968,167.325,54.162,160.046
C09695=1015.200,188.884,-127.990,167.329,54.151,160.044
C09696=1015.205,189.134,-128.011,167.333,54.141,160.043
C09697=1015.209,189.383,-128.033,167.338,54.129,160.042
C09698=1015.213,189.631,-128.054,167.342,54.118,160.040
C09699=1015.217,189.880,-128.076,167.347,54.107,160.039
C09700=1015.222,190.130,-128.097,167.351,54.096,160.038
C09701=1015.227,190.379,-128.119,167.356,54.085,160.037
C09702=1015.231,190.628,-128.142,167.360,54.074,160.035
C09703=1015.235,190.877,-128.163,167.364,54.062,160.034
C09704=1015.240,191.125,-128.184,167.368,54.052,160.032
C09705=1015.244,191.375,-128.206,167.373,54.040,160.031
C09706=1015.248,191.624,-128.228,167.377,54.029,160.030
C09707=1015.253,191.873,-128.250,167.382,54.019,160.029
C09708=1015.257,192.122,-128.271,167.387,54.007,160.027
C09709=1015.261,192.371,-128.293,167.391,53.996,160.026
C09710=1015.266,192.620,-128.314,167.395,53.985,160.025
C09711=1015.270,192.869,-128.336,167.399,53.974,160.023
C09712=1015.275,193.118,-128.358,167.405,53.963,160.022
C09713=1015.279,193.367,-128.380,167.409,53.952,160.021
C09714=1015.284,193.616,-128.402,167.413,53.941,160.019
C09715=1015.289,193.865,-128.424,167.418,53.930,160.018
C09716=1015.293,194.113,-128.445,167.422,53.919,160.017
C09717=1015.297,194.363,-128.467,167.426,53.907,160.015
C09718=1015.301,194.612,-128.489,167.432,53.897,160.014
C09719=1015.306,194.861,-128.510,167.436,53.885,160.013
C09720=1015.310,195.110,-128.532,167.440,53.874,160.011
C09721=1015.315,195.359,-128.554,167.445,53.863,160.010
C09722=1015.320,195.608,-128.576,167.450,53.852,160.009
C09723=1015.325,195.857,-128.598,167.455,53.841,160.008
C09724=1015.329,196.106,-128.620,167.459,53.830,160.006
C09725=1015.333,196.355,-128.641,167.463,53.819,160.005
C09726=1015.338,196.604,-128.663,167.469,53.808,160.004
C09727=1015.342,196.853,-128.686,167.473,53.797,160.002
C09728=1015.347,197.102,-128.708,167.478,53.785,160.001
C09729=1015.352,197.351,-128.729,167.482,53.775,160.000
C09730=1015.356,197.600,-128.751,167.486,53.764,159.999
C09731=1015.360,197.849,-128.773,167.491,53.752,159.997
C09732=1015.365,198.098,-128.795,167.496,53.742,159.996
C09733=1015.370,198.347,-128.817,167.501,53.730,159.995
C09734=1015.374,198.596,-128.839,167.505,53.719,159.993
C09735=1015.379,198.845,-128.861,167.511,53.708,159.992
C09736=1015.384,199.094,-128.883,167.515,53.697,159.991
C09737=1015.388,199.343,-128.905,167.519,53.686,159.990
C09738=1015.392,199.592,-128.928,167.524,53.675,159.988
C09739=1015.397,199.841,-128.950,167.529,53.664,159.987
C09740=1015.401,200.090,-128.972,167.533,53.653,159.986
C09741=1015.405,200.339,-128.995,167.538,53.642,159.985
C09742=1015.410,200.587,-129.017,167.543,53.631,159.983
C09743=1015.414,200.836,-129.040,167.547,53.621,159.982
C09744=1015.418,201.086,-129.062,167.552,53.609,159.981
C09745=1015.423,201.334,-129.084,167.557,53.599,159.980
C09746=1015.427,201.584,-129.107,167.562,53.587,159.978
C09747=1015.431,201.833,-129.129,167.566,53.577,159.977
C09748=1015.436,202.081,-129.152,167.571,53.567,159.976
C09749=1015.440,202.330,-129.174,167.576,53.555,159.975
C09750=1015.459,203.399,-129.271,168.088,53.620,160.098
C09751=1015.466,203.645,-129.294,168.093,53.610,160.097
C09752=1015.471,203.890,-129.318,168.096,53.600,160.095
C09753=1015.476,204.134,-129.342,168.100,53.591,160.094
C09754=1015.482,204.380,-129.366,168.105,53.581,160.093
C09755=1015.487,204.624,-129.390,168.109,53.572,160.092
C09756=1015.493,204.869,-129.413,168.114,53.561,160.090
C09757=1015.498,205.114,-129.437,168.118,53.552,160.089
C09758=1015.503,205.359,-129.461,168.122,53.543,160.088
C09759=1015.508,205.608,-129.486,168.126,53.533,160.087
C09760=1015.513,205.857,-129.509,168.130,53.524,160.086
C09761=1015.519,206.106,-129.534,168.134,53.514,160.085
C09762=1015.525,206.355,-129.557,168.139,53.504,160.084
C09763=1015.531,206.603,-129.582,168.143,53.495,160.082
C09764=1015.536,206.852,-129.606,168.148,53.485,160.081
C09765=1015.542,207.100,-129.631,168.152,53.476,160.080
C09766=1015.547,207.349,-129.655,168.156,53.466,160.079
C09767=1015.553,207.598,-129.680,168.161,53.457,160.078
C09768=1015.559,207.847,-129.704,168.165,53.448,160.077
C09769=1015.564,208.096,-129.729,168.168,53.438,160.075
C09770=1015.568,208.344,-129.753,168.173,53.428,160.074
C09771=1015.574,208.593,-129.778,168.177,53.419,160.073
C09772=1015.580,208.842,-129.802,168.181,53.409,160.072
C09773=1015.585,209.091,-129.827,168.186,53.400,160.071
C09774=1015.590,209.339,-129.851,168.190,53.390,160.070
C09775=1015.596,209.588,-129.876,168.194,53.381,160.069
C09776=1015.602,209.837,-129.900,168.199,53.371,160.068
C09777=1015.607,210.085,-129.925,168.203,53.363,160.067
C09778=1015.613,210.335,-129.949,168.207,53.354,160.066
C09779=1015.618,210.583,-129.975,168.211,53.344,160.064
C09780=1015.623,210.831,-129.999,168.216,53.335,160.063
C09781=1015.629,211.081,-130.024,168.220,53.325,160.062
C09782=1015.635,211.329,-130.049,168.224,53.316,160.061
C09783=1015.639,211.578,-130.074,168.229,53.308,160.060
C09784=1015.645,211.827,-130.098,168.233,53.298,160.059
C09785=1015.651,212.075,-130.123,168.238,53.289,160.058
C09786=1015.657,212.324,-130.148,168.242,53.280,160.057
C09787=1015.661,212.562,-130.172,168.246,53.271,160.056
C09788=1015.666,212.800,-130.195,168.250,53.262,160.055
C09789=1015.672,213.039,-130.219,168.253,53.254,160.054
C09790=1015.677,213.276,-130.243,168.258,53.245,160.053
C09791=1015.682,213.515,-130.267,168.262,53.236,160.052
C09792=1015.688,213.753,-130.290,168.266,53.227,160.051
C09793=1015.692,213.991,-130.314,168.271,53.219,160.050
C09794=1015.698,214.230,-130.338,168.275,53.209,160.049
C09795=1015.704,214.478,-130.363,168.279,53.201,160.048
C09796=1015.709,214.727,-130.388,168.283,53.192,160.046
C09797=1015.715,214.975,-130.413,168.288,53.183,160.046
C09798=1015.720,215.225,-130.438,168.292,53.174,160.044
C09799=1015.726,215.473,-130.463,168.296,53.165,160.043
C09800=1015.732,215.722,-130.487,168.301,53.156,160.042
C09801=1015.737,215.970,-130.513,168.305,53.146,160.041
C09802=1015.743,216.220,-130.537,168.309,53.137,160.040
C09803=1015.748,216.467,-130.562,168.314,53.129,160.039
C09804=1015.754,216.717,-130.587,168.318,53.119,160.038
C09805=1015.759,216.965,-130.613,168.322,53.111,160.037
C09806=1015.765,217.214,-130.637,168.326,53.102,160.036
C09807=1015.771,217.462,-130.662,168.331,53.093,160.035
C09808=1015.777,217.711,-130.688,168.336,53.084,160.034
C09809=1015.781,217.960,-130.712,168.340,53.075,160.033
C09810=1015.788,218.209,-130.738,168.344,53.066,160.032
C09811=1015.792,218.449,-130.762,168.348,53.058,160.031
C09812=1015.797,218.691,-130.786,168.352,53.049,160.030
C09813=1015.803,218.932,-130.811,168.357,53.041,160.029
C09814=1015.808,219.173,-130.836,168.361,53.032,160.028
C09815=1015.813,219.415,-130.861,168.365,53.024,160.027
C09816=1015.818,219.657,-130.885,168.369,53.016,160.026
C09817=1015.824,219.898,-130.910,168.374,53.007,160.025
C09818=1015.830,220.139,-130.934,168.378,52.999,160.024
C09819=1015.835,220.388,-130.960,168.383,52.990,160.023
C09820=1015.841,220.637,-130.986,168.387,52.982,160.022
C09821=1015.846,220.885,-131.011,168.391,52.972,160.021
C09822=1015.851,221.134,-131.036,168.396,52.964,160.020
C09823=1015.857,221.382,-131.061,168.400,52.955,160.019
C09824=1015.862,221.631,-131.087,168.404,52.947,160.018
C09825=1015.869,221.880,-131.112,168.408,52.939,160.017
C09826=1015.874,222.128,-131.138,168.412,52.930,160.016
C09827=1015.880,222.377,-131.163,168.417,52.921,160.015
C09828=1015.885,222.625,-131.189,168.421,52.913,160.014
C09829=1015.891,222.874,-131.214,168.426,52.904,160.013
C09830=1015.896,223.123,-131.239,168.430,52.896,160.013
C09831=1015.901,223.372,-131.265,168.435,52.887,160.012
C09832=1015.907,223.620,-131.290,168.439,52.879,160.011
C09833=1015.913,223.869,-131.316,168.444,52.870,160.010
C09834=1015.919,224.118,-131.341,168.448,52.862,160.009
C09835=1015.924,224.366,-131.367,168.453,52.853,160.008
C09836=1015.930,224.615,-131.392,168.457,52.844,160.007
C09837=1015.935,224.864,-131.418,168.462,52.836,160.006
C09838=1015.941,225.112,-131.443,168.466,52.827,160.005
C09839=1015.946,225.361,-131.469,168.470,52.819,160.004
C09840=1015.952,225.610,-131.495,168.474,52.810,160.003
C09841=1015.958,225.859,-131.520,168.479,52.802,160.002
C09842=1015.963,226.107,-131.546,168.483,52.794,160.001
C09843=1015.969,226.356,-131.571,168.488,52.786,160.000
C09844=1015.975,226.604,-131.598,168.493,52.777,159.999
C09845=1015.980,226.852,-131.623,168.497,52.769,159.999
C09846=1015.985,227.101,-131.649,168.501,52.761,159.998
C09847=1015.991,227.350,-131.675,168.505,52.752,159.997
C09848=1015.997,227.598,-131.701,168.510,52.744,159.996
C09849=1016.002,227.846,-131.727,168.515,52.736,159.995
C09850=1016.008,228.095,-131.753,168.519,52.728,159.994
C09851=1016.013,228.344,-131.779,168.523,52.719,159.993
C09852=1016.019,228.593,-131.805,168.527,52.711,159.992
C09853=1016.025,228.841,-131.831,168.532,52.703,159.991
C09854=1016.030,229.090,-131.856,168.537,52.695,159.990
C09855=1016.035,229.339,-131.882,168.542,52.686,159.990
C09856=1016.041,229.587,-131.909,168.546,52.679,159.989
C09857=1016.047,229.836,-131.935,168.550,52.671,159.988
C09858=1016.052,230.084,-131.962,168.555,52.662,159.987
C09859=1016.058,230.332,-131.986,168.559,52.655,159.986
C09860=1016.063,230.581,-132.012,168.563,52.646,159.985
C09861=1016.069,230.830,-132.039,168.568,52.639,159.984
C09862=1016.075,231.079,-132.065,168.573,52.630,159.984
C09863=1016.080,231.327,-132.092,168.577,52.623,159.983
C09864=1016.086,231.576,-132.118,168.581,52.614,159.982
C09865=1016.091,231.824,-132.144,168.586,52.607,159.981
C09866=1016.097,232.073,-132.170,168.590,52.598,159.980
C09867=1016.102,232.321,-132.196,168.595,52.591,159.979
C09868=1016.108,232.570,-132.222,168.599,52.582,159.978
C09869=1016.114,232.818,-132.249,168.603,52.575,159.978
C09870=1016.119,233.067,-132.275,168.608,52.566,159.977
C09871=1016.124,233.304,-132.300,168.613,52.559,159.976
C09872=1016.129,233.541,-132.325,168.617,52.551,159.975
C09873=1016.135,233.779,-132.350,168.621,52.544,159.974
C09874=1016.140,234.016,-132.376,168.625,52.537,159.974
C09875=1016.146,234.253,-132.400,168.630,52.529,159.973
C09876=1016.151,234.490,-132.426,168.634,52.522,159.972
C09877=1016.157,234.728,-132.451,168.638,52.514,159.971
C09878=1016.162,234.965,-132.476,168.643,52.506,159.971
C09879=1016.168,235.213,-132.502,168.647,52.498,159.969
C09880=1016.173,235.462,-132.529,168.652,52.491,159.969
C09881=1016.179,235.711,-132.555,168.656,52.482,159.968
C09882=1016.185,235.959,-132.582,168.660,52.475,159.967
C09883=1016.190,236.208,-132.608,168.665,52.467,159.966
C09884=1016.196,236.457,-132.634,168.670,52.459,159.966
C09885=1016.202,236.705,-132.661,168.674,52.451,159.965
C09886=1016.207,236.953,-132.688,168.679,52.444,159.964
C09887=1016.213,237.202,-132.714,168.683,52.436,159.963
C09888=1016.219,237.451,-132.740,168.688,52.429,159.962
C09889=1016.224,237.699,-132.767,168.693,52.420,159.961
C09890=1016.230,237.947,-132.793,168.697,52.413,159.961
C09891=1016.236,238.196,-132.820,168.702,52.405,159.960
C09892=1016.242,238.444,-132.847,168.707,52.397,159.959
C09893=1016.247,238.693,-132.873,168.711,52.390,159.958
C09894=1016.253,238.941,-132.899,168.716,52.382,159.958
C09895=1016.258,239.190,-132.927,168.720,52.375,159.957
C09896=1016.264,239.438,-132.953,168.725,52.367,159.956
C09897=1016.270,239.687,-132.980,168.729,52.360,159.955
C09898=1016.275,239.935,-133.007,168.734,52.352,159.955
C09899=1016.280,240.184,-133.034,168.738,52.345,159.954
C09900=1016.286,240.432,-133.060,168.743,52.337,159.953
C09901=1016.291,240.681,-133.088,168.747,52.330,159.952
C09902=1016.297,240.929,-133.114,168.752,52.322,159.952
C09903=1016.303,241.178,-133.141,168.756,52.315,159.951
C09904=1016.308,241.427,-133.168,168.761,52.307,159.950
C09905=1016.314,241.675,-133.196,168.765,52.300,159.949
C09906=1016.320,241.923,-133.223,168.770,52.292,159.949
C09907=1016.326,242.171,-133.249,168.774,52.285,159.948
C09908=1016.331,242.420,-133.276,168.780,52.277,159.947
C09909=1016.337,242.668,-133.303,168.784,52.270,159.946
C09910=1016.343,242.917,-133.330,168.789,52.263,159.946
C09911=1016.348,243.165,-133.358,168.793,52.256,159.945
C09912=1016.353,243.413,-133.385,168.798,52.248,159.944
C09913=1016.359,243.662,-133.412,168.803,52.241,159.944
C09914=1016.364,243.911,-133.439,168.807,52.234,159.943
C09915=1016.370,244.159,-133.467,168.812,52.226,159.942
C09916=1016.375,244.408,-133.494,168.816,52.219,159.941
C09917=1016.380,244.656,-133.521,168.821,52.212,159.941
C09918=1016.387,244.904,-133.548,168.825,52.205,159.940
C09919=1016.392,245.153,-133.576,168.830,52.198,159.940
C09920=1016.398,245.402,-133.603,168.835,52.190,159.939
C09921=1016.403,245.650,-133.631,168.839,52.183,159.938
C09922=1016.408,245.898,-133.658,168.845,52.176,159.938
C09923=1016.414,246.146,-133.685,168.849,52.169,159.937
C09924=1016.419,246.395,-133.712,168.853,52.162,159.936
C09925=1016.426,246.644,-133.739,168.858,52.154,159.935
C09926=1016.431,246.892,-133.767,168.863,52.148,159.935
C09927=1016.436,247.141,-133.795,168.867,52.141,159.934
C09928=1016.442,247.388,-133.822,168.872,52.133,159.933
C09929=1016.448,247.638,-133.850,168.876,52.126,159.933
C09930=1016.454,247.885,-133.877,168.881,52.119,159.932
C09931=1016.459,248.120,-133.903,168.885,52.112,159.931
C09932=1016.464,248.353,-133.929,168.889,52.106,159.931
C09933=1016.470,248.587,-133.954,168.894,52.099,159.930
C09934=1016.475,248.820,-133.980,168.898,52.093,159.930
C09935=1016.480,249.055,-134.006,168.903,52.086,159.929
C09936=1016.486,249.288,-134.032,168.907,52.079,159.928
C09937=1016.491,249.522,-134.058,168.912,52.073,159.928
C09938=1016.496,249.756,-134.085,168.916,52.066,159.927
C09939=1016.502,250.004,-134.112,168.921,52.060,159.927
C09940=1016.507,250.252,-134.139,168.926,52.052,159.926
C09941=1016.514,250.502,-134.167,168.931,52.045,159.925
C09942=1016.519,250.750,-134.194,168.935,52.038,159.924
C09943=1016.525,250.998,-134.222,168.940,52.031,159.924
C09944=1016.531,251.247,-134.249,168.945,52.024,159.923
C09945=1016.536,251.495,-134.277,168.949,52.017,159.923
C09946=1016.542,251.742,-134.305,168.954,52.010,159.922
C09947=1016.548,251.992,-134.332,168.959,52.004,159.921
C09948=1016.553,252.240,-134.360,168.963,51.996,159.921
C09949=1016.560,252.488,-134.388,168.968,51.989,159.920
C09950=1016.565,252.737,-134.415,168.973,51.983,159.920
C09951=1016.571,252.986,-134.444,168.977,51.976,159.919
C09952=1016.577,253.234,-134.471,168.983,51.969,159.918
C09953=1016.582,253.482,-134.499,168.987,51.962,159.918
C09954=1016.589,253.731,-134.526,168.992,51.955,159.917
C09955=1016.594,253.979,-134.554,168.997,51.948,159.917
C09956=1016.600,254.227,-134.582,169.002,51.942,159.916
C09957=1016.606,254.475,-134.610,169.006,51.935,159.915
C09958=1016.612,254.725,-134.637,169.011,51.928,159.915
C09959=1016.617,254.973,-134.665,169.016,51.921,159.914
C09960=1016.624,255.221,-134.693,169.020,51.914,159.913
C09961=1016.629,255.469,-134.721,169.026,51.908,159.913
C09962=1016.636,255.718,-134.749,169.030,51.901,159.912
C09963=1016.641,255.966,-134.777,169.035,51.894,159.912
C09964=1016.647,256.214,-134.805,169.040,51.887,159.911
C09965=1016.653,256.463,-134.832,169.045,51.880,159.910
C09966=1016.659,256.711,-134.860,169.049,51.874,159.910
C09967=1016.665,256.960,-134.888,169.055,51.867,159.909
C09968=1016.671,257.208,-134.916,169.059,51.860,159.909
C09969=1016.677,257.457,-134.944,169.064,51.854,159.908
C09970=1016.683,257.704,-134.971,169.069,51.847,159.908
C09971=1016.689,257.953,-135.000,169.074,51.840,159.907
C09972=1016.694,258.201,-135.028,169.078,51.833,159.906
C09973=1016.701,258.450,-135.055,169.083,51.827,159.906
C09974=1016.707,258.698,-135.084,169.088,51.820,159.905
C09975=1016.712,258.946,-135.112,169.093,51.813,159.905
C09976=1016.719,259.195,-135.139,169.097,51.807,159.904
C09977=1016.725,259.444,-135.168,169.103,51.800,159.904
C09978=1016.731,259.691,-135.195,169.108,51.793,159.903
C09979=1016.737,259.940,-135.223,169.112,51.788,159.903
C09980=1016.742,260.188,-135.253,169.117,51.781,159.902
C09981=1016.748,260.437,-135.281,169.122,51.774,159.902
C09982=1016.754,260.685,-135.309,169.127,51.767,159.901
C09983=1016.759,260.933,-135.338,169.132,51.762,159.901
C09984=1016.765,261.182,-135.366,169.137,51.755,159.900
C09985=1016.771,261.430,-135.395,169.141,51.748,159.899
C09986=1016.777,261.678,-135.423,169.146,51.743,159.899
C09987=1016.783,261.927,-135.452,169.152,51.736,159.899
C09988=1016.789,262.175,-135.480,169.156,51.729,159.898
C09989=1016.794,262.423,-135.509,169.161,51.723,159.898
C09990=1016.800,262.671,-135.537,169.166,51.717,159.897
C09991=1016.806,262.904,-135.564,169.171,51.711,159.897
C09992=1016.811,263.138,-135.590,169.176,51.705,159.896
C09993=1016.817,263.370,-135.617,169.179,51.699,159.896
C09994=1016.822,263.603,-135.644,169.184,51.693,159.895
C09995=1016.828,263.835,-135.671,169.189,51.687,159.895
C09996=1016.833,264.069,-135.698,169.193,51.682,159.894
//INST
///DATE 2021/06/17 10:59
///ATTR SC,RW,RJ
////FRAME ROBOT
///GROUP1 RB1
NOP
MOVL C00000 V=800.0 PL=0
MOVL C00001 V=800.0 PL=0
MOVL C00002 V=800.0 PL=0
MOVL C00003 V=800.0 PL=0
MOVL C00004 V=800.0 PL=0
MOVL C00005 V=800.0 PL=0
MOVL C00006 V=800.0 PL=0
MOVL C00007 V=800.0 PL=0
MOVL C00008 V=800.0 PL=0
MOVL C00009 V=800.0 PL=0
MOVL C00010 V=800.0 PL=0
MOVL C00011 V=800.0 PL=0
MOVL C00012 V=800.0 PL=0
MOVL C00013 V=800.0 PL=0
MOVL C00014 V=800.0 PL=0
MOVL C00015 V=800.0 PL=0
MOVL C00016 V=800.0 PL=0
MOVL C00017 V=800.0 PL=0
MOVL C00018 V=800.0 PL=0
MOVL C00019 V=800.0 PL=0
MOVL C00020 V=800.0 PL=0
MOVL C00021 V=800.0 PL=0
MOVL C00022 V=800.0 PL=0
MOVL C00023 V=800.0 PL=0
MOVL C00024 V=800.0 PL=0
MOVL C00025 V=800.0 PL=0
MOVL C00026 V=800.0 PL=0
MOVL C00027 V=800.0 PL=0
MOVL C00028 V=800.0 PL=0
MOVL C00029 V=800.0 PL=0
MOVL C00030 V=800.0 PL=0
MOVL C00031 V=800.0 PL=0
MOVL C00032 V=800.0 PL=0
MOVL C00033 V=800.0 PL=0
MOVL C00034 V=800.0 PL=0
MOVL C00035 V=800.0 PL=0
MOVL C00036 V=800.0 PL=0
MOVL C00037 V=800.0 PL=0
MOVL C00038 V=800.0 PL=0
MOVL C00039 V=800.0 PL=0
MOVL C00040 V=800.0 PL=0
MOVL C00041 V=800.0 PL=0
MOVL C00042 V=800.0 PL=0
MOVL C00043 V=800.0 PL=0
MOVL C00044 V=800.0 PL=0
MOVL C00045 V=800.0 PL=0
MOVL C00046 V=800.0 PL=0
MOVL C00047 V=800.0 PL=0
MOVL C00048 V=800.0 PL=0
MOVL C00049 V=800.0 PL=0
MOVL C00050 V=800.0 PL=0
MOVL C00051 V=800.0 PL=0
MOVL C00052 V=800.0 PL=0
MOVL C00053 V=800.0 PL=0
MOVL C00054 V=800.0 PL=0
MOVL C00055 V=800.0 PL=0
MOVL C00056 V=800.0 PL=0
MOVL C00057 V=800.0 PL=0
MOVL C00058 V=800.0 PL=0
MOVL C00059 V=800.0 PL=0
MOVL C00060 V=800.0 PL=0
MOVL C00061 V=800.0 PL=0
MOVL C00062 V=800.0 PL=0
MOVL C00063 V=800.0 PL=0
MOVL C00064 V=800.0 PL=0
MOVL C00065 V=800.0 PL=0
MOVL C00066 V=800.0 PL=0
MOVL C00067 V=800.0 PL=0
MOVL C00068 V=800.0 PL=0
MOVL C00069 V=800.0 PL=0
MOVL C00070 V=800.0 PL=0
MOVL C00071 V=800.0 PL=0
MOVL C00072 V=800.0 PL=0
MOVL C00073 V=800.0 PL=0
MOVL C00074 V=800.0 PL=0
MOVL C00075 V=800.0 PL=0
MOVL C00076 V=800.0 PL=0
MOVL C00077 V=800.0 PL=0
MOVL C00078 V=800.0 PL=0
MOVL C00079 V=800.0 PL=0
MOVL C00080 V=800.0 PL=0
MOVL C00081 V=800.0 PL=0
MOVL C00082 V=800.0 PL=0
MOVL C00083 V=800.0 PL=0
MOVL C00084 V=800.0 PL=0
MOVL C00085 V=800.0 PL=0
MOVL C00086 V=800.0 PL=0
MOVL C00087 V=800.0 PL=0
MOVL C00088 V=800.0 PL=0
MOVL C00089 V=800.0 PL=0
MOVL C00090 V=800.0 PL=0
MOVL C00091 V=800.0 PL=0
MOVL C00092 V=800.0 PL=0
MOVL C00093 V=800.0 PL=0
MOVL C00094 V=800.0 PL=0
MOVL C00095 V=800.0 PL=0
MOVL C00096 V=800.0 PL=0
MOVL C00097 V=800.0 PL=0
MOVL C00098 V=800.0 PL=0
MOVL C00099 V=800.0 PL=0
MOVL C00100 V=800.0 PL=0
MOVL C00101 V=800.0 PL=0
MOVL C00102 V=800.0 PL=0
MOVL C00103 V=800.0 PL=0
MOVL C00104 V=800.0 PL=0
MOVL C00105 V=800.0 PL=0
MOVL C00106 V=800.0 PL=0
MOVL C00107 V=800.0 PL=0
MOVL C00108 V=800.0 PL=0
MOVL C00109 V=800.0 PL=0
MOVL C00110 V=800.0 PL=0
MOVL C00111 V=800.0 PL=0
MOVL C00112 V=800.0 PL=0
MOVL C00113 V=800.0 PL=0
MOVL C00114 V=800.0 PL=0
MOVL C00115 V=800.0 PL=0
MOVL C00116 V=800.0 PL=0
MOVL C00117 V=800.0 PL=0
MOVL C00118 V=800.0 PL=0
MOVL C00119 V=800.0 PL=0
MOVL C00120 V=800.0 PL=0
MOVL C00121 V=800.0 PL=0
MOVL C00122 V=800.0 PL=0
MOVL C00123 V=800.0 PL=0
MOVL C00124 V=800.0 PL=0
MOVL C00125 V=800.0 PL=0
MOVL C00126 V=800.0 PL=0
MOVL C00127 V=800.0 PL=0
MOVL C00128 V=800.0 PL=0
MOVL C00129 V=800.0 PL=0
MOVL C00130 V=800.0 PL=0
MOVL C00131 V=800.0 PL=0
MOVL C00132 V=800.0 PL=0
MOVL C00133 V=800.0 PL=0
MOVL C00134 V=800.0 PL=0
MOVL C00135 V=800.0 PL=0
MOVL C00136 V=800.0 PL=0
MOVL C00137 V=800.0 PL=0
MOVL C00138 V=800.0 PL=0
MOVL C00139 V=800.0 PL=0
MOVL C00140 V=800.0 PL=0
MOVL C00141 V=800.0 PL=0
MOVL C00142 V=800.0 PL=0
MOVL C00143 V=800.0 PL=0
MOVL C00144 V=800.0 PL=0
MOVL C00145 V=800.0 PL=0
MOVL C00146 V=800.0 PL=0
MOVL C00147 V=800.0 PL=0
MOVL C00148 V=800.0 PL=0
MOVL C00149 V=800.0 PL=0
MOVL C00150 V=800.0 PL=0
MOVL C00151 V=800.0 PL=0
MOVL C00152 V=800.0 PL=0
MOVL C00153 V=800.0 PL=0
MOVL C00154 V=800.0 PL=0
MOVL C00155 V=800.0 PL=0
MOVL C00156 V=800.0 PL=0
MOVL C00157 V=800.0 PL=0
MOVL C00158 V=800.0 PL=0
MOVL C00159 V=800.0 PL=0
MOVL C00160 V=800.0 PL=0
MOVL C00161 V=800.0 PL=0
MOVL C00162 V=800.0 PL=0
MOVL C00163 V=800.0 PL=0
MOVL C00164 V=800.0 PL=0
MOVL C00165 V=800.0 PL=0
MOVL C00166 V=800.0 PL=0
MOVL C00167 V=800.0 PL=0
MOVL C00168 V=800.0 PL=0
MOVL C00169 V=800.0 PL=0
MOVL C00170 V=800.0 PL=0
MOVL C00171 V=800.0 PL=0
MOVL C00172 V=800.0 PL=0
MOVL C00173 V=800.0 PL=0
MOVL C00174 V=800.0 PL=0
MOVL C00175 V=800.0 PL=0
MOVL C00176 V=800.0 PL=0
MOVL C00177 V=800.0 PL=0
MOVL C00178 V=800.0 PL=0
MOVL C00179 V=800.0 PL=0
MOVL C00180 V=800.0 PL=0
MOVL C00181 V=800.0 PL=0
MOVL C00182 V=800.0 PL=0
MOVL C00183 V=800.0 PL=0
MOVL C00184 V=800.0 PL=0
MOVL C00185 V=800.0 PL=0
MOVL C00186 V=800.0 PL=0
MOVL C00187 V=800.0 PL=0
MOVL C00188 V=800.0 PL=0
MOVL C00189 V=800.0 PL=0
MOVL C00190 V=800.0 PL=0
MOVL C00191 V=800.0 PL=0
MOVL C00192 V=800.0 PL=0
MOVL C00193 V=800.0 PL=0
MOVL C00194 V=800.0 PL=0
MOVL C00195 V=800.0 PL=0
MOVL C00196 V=800.0 PL=0
MOVL C00197 V=800.0 PL=0
MOVL C00198 V=800.0 PL=0
MOVL C00199 V=800.0 PL=0
MOVL C00200 V=800.0 PL=0
MOVL C00201 V=800.0 PL=0
MOVL C00202 V=800.0 PL=0
MOVL C00203 V=800.0 PL=0
MOVL C00204 V=800.0 PL=0
MOVL C00205 V=800.0 PL=0
MOVL C00206 V=800.0 PL=0
MOVL C00207 V=800.0 PL=0
MOVL C00208 V=800.0 PL=0
MOVL C00209 V=800.0 PL=0
MOVL C00210 V=800.0 PL=0
MOVL C00211 V=800.0 PL=0
MOVL C00212 V=800.0 PL=0
MOVL C00213 V=800.0 PL=0
MOVL C00214 V=800.0 PL=0
MOVL C00215 V=800.0 PL=0
MOVL C00216 V=800.0 PL=0
MOVL C00217 V=800.0 PL=0
MOVL C00218 V=800.0 PL=0
MOVL C00219 V=800.0 PL=0
MOVL C00220 V=800.0 PL=0
MOVL C00221 V=800.0 PL=0
MOVL C00222 V=800.0 PL=0
MOVL C00223 V=800.0 PL=0
MOVL C00224 V=800.0 PL=0
MOVL C00225 V=800.0 PL=0
MOVL C00226 V=800.0 PL=0
MOVL C00227 V=800.0 PL=0
MOVL C00228 V=800.0 PL=0
MOVL C00229 V=800.0 PL=0
MOVL C00230 V=800.0 PL=0
MOVL C00231 V=800.0 PL=0
MOVL C00232 V=800.0 PL=0
MOVL C00233 V=800.0 PL=0
MOVL C00234 V=800.0 PL=0
MOVL C00235 V=800.0 PL=0
MOVL C00236 V=800.0 PL=0
MOVL C00237 V=800.0 PL=0
MOVL C00238 V=800.0 PL=0
MOVL C00239 V=800.0 PL=0
MOVL C00240 V=800.0 PL=0
MOVL C00241 V=800.0 PL=0
MOVL C00242 V=800.0 PL=0
MOVL C00243 V=800.0 PL=0
MOVL C00244 V=800.0 PL=0
MOVL C00245 V=800.0 PL=0
MOVL C00246 V=800.0 PL=0
MOVL C00247 V=800.0 PL=0
MOVL C00248 V=800.0 PL=0
MOVL C00249 V=800.0 PL=0
MOVL C00250 V=800.0 PL=0
MOVL C00251 V=800.0 PL=0
MOVL C00252 V=800.0 PL=0
MOVL C00253 V=800.0 PL=0
MOVL C00254 V=800.0 PL=0
MOVL C00255 V=800.0 PL=0
MOVL C00256 V=800.0 PL=0
MOVL C00257 V=800.0 PL=0
MOVL C00258 V=800.0 PL=0
MOVL C00259 V=800.0 PL=0
MOVL C00260 V=800.0 PL=0
MOVL C00261 V=800.0 PL=0
MOVL C00262 V=800.0 PL=0
MOVL C00263 V=800.0 PL=0
MOVL C00264 V=800.0 PL=0
MOVL C00265 V=800.0 PL=0
MOVL C00266 V=800.0 PL=0
MOVL C00267 V=800.0 PL=0
MOVL C00268 V=800.0 PL=0
MOVL C00269 V=800.0 PL=0
MOVL C00270 V=800.0 PL=0
MOVL C00271 V=800.0 PL=0
MOVL C00272 V=800.0 PL=0
MOVL C00273 V=800.0 PL=0
MOVL C00274 V=800.0 PL=0
MOVL C00275 V=800.0 PL=0
MOVL C00276 V=800.0 PL=0
MOVL C00277 V=800.0 PL=0
MOVL C00278 V=800.0 PL=0
MOVL C00279 V=800.0 PL=0
MOVL C00280 V=800.0 PL=0
MOVL C00281 V=800.0 PL=0
MOVL C00282 V=800.0 PL=0
MOVL C00283 V=800.0 PL=0
MOVL C00284 V=800.0 PL=0
MOVL C00285 V=800.0 PL=0
MOVL C00286 V=800.0 PL=0
MOVL C00287 V=800.0 PL=0
MOVL C00288 V=800.0 PL=0
MOVL C00289 V=800.0 PL=0
MOVL C00290 V=800.0 PL=0
MOVL C00291 V=800.0 PL=0
MOVL C00292 V=800.0 PL=0
MOVL C00293 V=800.0 PL=0
MOVL C00294 V=800.0 PL=0
MOVL C00295 V=800.0 PL=0
MOVL C00296 V=800.0 PL=0
MOVL C00297 V=800.0 PL=0
MOVL C00298 V=800.0 PL=0
MOVL C00299 V=800.0 PL=0
MOVL C00300 V=800.0 PL=0
MOVL C00301 V=800.0 PL=0
MOVL C00302 V=800.0 PL=0
MOVL C00303 V=800.0 PL=0
MOVL C00304 V=800.0 PL=0
MOVL C00305 V=800.0 PL=0
MOVL C00306 V=800.0 PL=0
MOVL C00307 V=800.0 PL=0
MOVL C00308 V=800.0 PL=0
MOVL C00309 V=800.0 PL=0
MOVL C00310 V=800.0 PL=0
MOVL C00311 V=800.0 PL=0
MOVL C00312 V=800.0 PL=0
MOVL C00313 V=800.0 PL=0
MOVL C00314 V=800.0 PL=0
MOVL C00315 V=800.0 PL=0
MOVL C00316 V=800.0 PL=0
MOVL C00317 V=800.0 PL=0
MOVL C00318 V=800.0 PL=0
MOVL C00319 V=800.0 PL=0
MOVL C00320 V=800.0 PL=0
MOVL C00321 V=800.0 PL=0
MOVL C00322 V=800.0 PL=0
MOVL C00323 V=800.0 PL=0
MOVL C00324 V=800.0 PL=0
MOVL C00325 V=800.0 PL=0
MOVL C00326 V=800.0 PL=0
MOVL C00327 V=800.0 PL=0
MOVL C00328 V=800.0 PL=0
MOVL C00329 V=800.0 PL=0
MOVL C00330 V=800.0 PL=0
MOVL C00331 V=800.0 PL=0
MOVL C00332 V=800.0 PL=0
MOVL C00333 V=800.0 PL=0
MOVL C00334 V=800.0 PL=0
MOVL C00335 V=800.0 PL=0
MOVL C00336 V=800.0 PL=0
MOVL C00337 V=800.0 PL=0
MOVL C00338 V=800.0 PL=0
MOVL C00339 V=800.0 PL=0
MOVL C00340 V=800.0 PL=0
MOVL C00341 V=800.0 PL=0
MOVL C00342 V=800.0 PL=0
MOVL C00343 V=800.0 PL=0
MOVL C00344 V=800.0 PL=0
MOVL C00345 V=800.0 PL=0
MOVL C00346 V=800.0 PL=0
MOVL C00347 V=800.0 PL=0
MOVL C00348 V=800.0 PL=0
MOVL C00349 V=800.0 PL=0
MOVL C00350 V=800.0 PL=0
MOVL C00351 V=800.0 PL=0
MOVL C00352 V=800.0 PL=0
MOVL C00353 V=800.0 PL=0
MOVL C00354 V=800.0 PL=0
MOVL C00355 V=800.0 PL=0
MOVL C00356 V=800.0 PL=0
MOVL C00357 V=800.0 PL=0
MOVL C00358 V=800.0 PL=0
MOVL C00359 V=800.0 PL=0
MOVL C00360 V=800.0 PL=0
MOVL C00361 V=800.0 PL=0
MOVL C00362 V=800.0 PL=0
MOVL C00363 V=800.0 PL=0
MOVL C00364 V=800.0 PL=0
MOVL C00365 V=800.0 PL=0
MOVL C00366 V=800.0 PL=0
MOVL C00367 V=800.0 PL=0
MOVL C00368 V=800.0 PL=0
MOVL C00369 V=800.0 PL=0
MOVL C00370 V=800.0 PL=0
MOVL C00371 V=800.0 PL=0
MOVL C00372 V=800.0 PL=0
MOVL C00373 V=800.0 PL=0
MOVL C00374 V=800.0 PL=0
MOVL C00375 V=800.0 PL=0
MOVL C00376 V=800.0 PL=0
MOVL C00377 V=800.0 PL=0
MOVL C00378 V=800.0 PL=0
MOVL C00379 V=800.0 PL=0
MOVL C00380 V=800.0 PL=0
MOVL C00381 V=800.0 PL=0
MOVL C00382 V=800.0 PL=0
MOVL C00383 V=800.0 PL=0
MOVL C00384 V=800.0 PL=0
MOVL C00385 V=800.0 PL=0
MOVL C00386 V=800.0 PL=0
MOVL C00387 V=800.0 PL=0
MOVL C00388 V=800.0 PL=0
MOVL C00389 V=800.0 PL=0
MOVL C00390 V=800.0 PL=0
MOVL C00391 V=800.0 PL=0
MOVL C00392 V=800.0 PL=0
MOVL C00393 V=800.0 PL=0
MOVL C00394 V=800.0 PL=0
MOVL C00395 V=800.0 PL=0
MOVL C00396 V=800.0 PL=0
MOVL C00397 V=800.0 PL=0
MOVL C00398 V=800.0 PL=0
MOVL C00399 V=800.0 PL=0
MOVL C00400 V=800.0 PL=0
MOVL C00401 V=800.0 PL=0
MOVL C00402 V=800.0 PL=0
MOVL C00403 V=800.0 PL=0
MOVL C00404 V=800.0 PL=0
MOVL C00405 V=800.0 PL=0
MOVL C00406 V=800.0 PL=0
MOVL C00407 V=800.0 PL=0
MOVL C00408 V=800.0 PL=0
MOVL C00409 V=800.0 PL=0
MOVL C00410 V=800.0 PL=0
MOVL C00411 V=800.0 PL=0
MOVL C00412 V=800.0 PL=0
MOVL C00413 V=800.0 PL=0
MOVL C00414 V=800.0 PL=0
MOVL C00415 V=800.0 PL=0
MOVL C00416 V=800.0 PL=0
MOVL C00417 V=800.0 PL=0
MOVL C00418 V=800.0 PL=0
MOVL C00419 V=800.0 PL=0
MOVL C00420 V=800.0 PL=0
MOVL C00421 V=800.0 PL=0
MOVL C00422 V=800.0 PL=0
MOVL C00423 V=800.0 PL=0
MOVL C00424 V=800.0 PL=0
MOVL C00425 V=800.0 PL=0
MOVL C00426 V=800.0 PL=0
MOVL C00427 V=800.0 PL=0
MOVL C00428 V=800.0 PL=0
MOVL C00429 V=800.0 PL=0
MOVL C00430 V=800.0 PL=0
MOVL C00431 V=800.0 PL=0
MOVL C00432 V=800.0 PL=0
MOVL C00433 V=800.0 PL=0
MOVL C00434 V=800.0 PL=0
MOVL C00435 V=800.0 PL=0
MOVL C00436 V=800.0 PL=0
MOVL C00437 V=800.0 PL=0
MOVL C00438 V=800.0 PL=0
MOVL C00439 V=800.0 PL=0
MOVL C00440 V=800.0 PL=0
MOVL C00441 V=800.0 PL=0
MOVL C00442 V=800.0 PL=0
MOVL C00443 V=800.0 PL=0
MOVL C00444 V=800.0 PL=0
MOVL C00445 V=800.0 PL=0
MOVL C00446 V=800.0 PL=0
MOVL C00447 V=800.0 PL=0
MOVL C00448 V=800.0 PL=0
MOVL C00449 V=800.0 PL=0
MOVL C00450 V=800.0 PL=0
MOVL C00451 V=800.0 PL=0
MOVL C00452 V=800.0 PL=0
MOVL C00453 V=800.0 PL=0
MOVL C00454 V=800.0 PL=0
MOVL C00455 V=800.0 PL=0
MOVL C00456 V=800.0 PL=0
MOVL C00457 V=800.0 PL=0
MOVL C00458 V=800.0 PL=0
MOVL C00459 V=800.0 PL=0
MOVL C00460 V=800.0 PL=0
MOVL C00461 V=800.0 PL=0
MOVL C00462 V=800.0 PL=0
MOVL C00463 V=800.0 PL=0
MOVL C00464 V=800.0 PL=0
MOVL C00465 V=800.0 PL=0
MOVL C00466 V=800.0 PL=0
MOVL C00467 V=800.0 PL=0
MOVL C00468 V=800.0 PL=0
MOVL C00469 V=800.0 PL=0
MOVL C00470 V=800.0 PL=0
MOVL C00471 V=800.0 PL=0
MOVL C00472 V=800.0 PL=0
MOVL C00473 V=800.0 PL=0
MOVL C00474 V=800.0 PL=0
MOVL C00475 V=800.0 PL=0
MOVL C00476 V=800.0 PL=0
MOVL C00477 V=800.0 PL=0
MOVL C00478 V=800.0 PL=0
MOVL C00479 V=800.0 PL=0
MOVL C00480 V=800.0 PL=0
MOVL C00481 V=800.0 PL=0
MOVL C00482 V=800.0 PL=0
MOVL C00483 V=800.0 PL=0
MOVL C00484 V=800.0 PL=0
MOVL C00485 V=800.0 PL=0
MOVL C00486 V=800.0 PL=0
MOVL C00487 V=800.0 PL=0
MOVL C00488 V=800.0 PL=0
MOVL C00489 V=800.0 PL=0
MOVL C00490 V=800.0 PL=0
MOVL C00491 V=800.0 PL=0
MOVL C00492 V=800.0 PL=0
MOVL C00493 V=800.0 PL=0
MOVL C00494 V=800.0 PL=0
MOVL C00495 V=800.0 PL=0
MOVL C00496 V=800.0 PL=0
MOVL C00497 V=800.0 PL=0
MOVL C00498 V=800.0 PL=0
MOVL C00499 V=800.0 PL=0
MOVL C00500 V=800.0 PL=0
MOVL C00501 V=800.0 PL=0
MOVL C00502 V=800.0 PL=0
MOVL C00503 V=800.0 PL=0
MOVL C00504 V=800.0 PL=0
MOVL C00505 V=800.0 PL=0
MOVL C00506 V=800.0 PL=0
MOVL C00507 V=800.0 PL=0
MOVL C00508 V=800.0 PL=0
MOVL C00509 V=800.0 PL=0
MOVL C00510 V=800.0 PL=0
MOVL C00511 V=800.0 PL=0
MOVL C00512 V=800.0 PL=0
MOVL C00513 V=800.0 PL=0
MOVL C00514 V=800.0 PL=0
MOVL C00515 V=800.0 PL=0
MOVL C00516 V=800.0 PL=0
MOVL C00517 V=800.0 PL=0
MOVL C00518 V=800.0 PL=0
MOVL C00519 V=800.0 PL=0
MOVL C00520 V=800.0 PL=0
MOVL C00521 V=800.0 PL=0
MOVL C00522 V=800.0 PL=0
MOVL C00523 V=800.0 PL=0
MOVL C00524 V=800.0 PL=0
MOVL C00525 V=800.0 PL=0
MOVL C00526 V=800.0 PL=0
MOVL C00527 V=800.0 PL=0
MOVL C00528 V=800.0 PL=0
MOVL C00529 V=800.0 PL=0
MOVL C00530 V=800.0 PL=0
MOVL C00531 V=800.0 PL=0
MOVL C00532 V=800.0 PL=0
MOVL C00533 V=800.0 PL=0
MOVL C00534 V=800.0 PL=0
MOVL C00535 V=800.0 PL=0
MOVL C00536 V=800.0 PL=0
MOVL C00537 V=800.0 PL=0
MOVL C00538 V=800.0 PL=0
MOVL C00539 V=800.0 PL=0
MOVL C00540 V=800.0 PL=0
MOVL C00541 V=800.0 PL=0
MOVL C00542 V=800.0 PL=0
MOVL C00543 V=800.0 PL=0
MOVL C00544 V=800.0 PL=0
MOVL C00545 V=800.0 PL=0
MOVL C00546 V=800.0 PL=0
MOVL C00547 V=800.0 PL=0
MOVL C00548 V=800.0 PL=0
MOVL C00549 V=800.0 PL=0
MOVL C00550 V=800.0 PL=0
MOVL C00551 V=800.0 PL=0
MOVL C00552 V=800.0 PL=0
MOVL C00553 V=800.0 PL=0
MOVL C00554 V=800.0 PL=0
MOVL C00555 V=800.0 PL=0
MOVL C00556 V=800.0 PL=0
MOVL C00557 V=800.0 PL=0
MOVL C00558 V=800.0 PL=0
MOVL C00559 V=800.0 PL=0
MOVL C00560 V=800.0 PL=0
MOVL C00561 V=800.0 PL=0
MOVL C00562 V=800.0 PL=0
MOVL C00563 V=800.0 PL=0
MOVL C00564 V=800.0 PL=0
MOVL C00565 V=800.0 PL=0
MOVL C00566 V=800.0 PL=0
MOVL C00567 V=800.0 PL=0
MOVL C00568 V=800.0 PL=0
MOVL C00569 V=800.0 PL=0
MOVL C00570 V=800.0 PL=0
MOVL C00571 V=800.0 PL=0
MOVL C00572 V=800.0 PL=0
MOVL C00573 V=800.0 PL=0
MOVL C00574 V=800.0 PL=0
MOVL C00575 V=800.0 PL=0
MOVL C00576 V=800.0 PL=0
MOVL C00577 V=800.0 PL=0
MOVL C00578 V=800.0 PL=0
MOVL C00579 V=800.0 PL=0
MOVL C00580 V=800.0 PL=0
MOVL C00581 V=800.0 PL=0
MOVL C00582 V=800.0 PL=0
MOVL C00583 V=800.0 PL=0
MOVL C00584 V=800.0 PL=0
MOVL C00585 V=800.0 PL=0
MOVL C00586 V=800.0 PL=0
MOVL C00587 V=800.0 PL=0
MOVL C00588 V=800.0 PL=0
MOVL C00589 V=800.0 PL=0
MOVL C00590 V=800.0 PL=0
MOVL C00591 V=800.0 PL=0
MOVL C00592 V=800.0 PL=0
MOVL C00593 V=800.0 PL=0
MOVL C00594 V=800.0 PL=0
MOVL C00595 V=800.0 PL=0
MOVL C00596 V=800.0 PL=0
MOVL C00597 V=800.0 PL=0
MOVL C00598 V=800.0 PL=0
MOVL C00599 V=800.0 PL=0
MOVL C00600 V=800.0 PL=0
MOVL C00601 V=800.0 PL=0
MOVL C00602 V=800.0 PL=0
MOVL C00603 V=800.0 PL=0
MOVL C00604 V=800.0 PL=0
MOVL C00605 V=800.0 PL=0
MOVL C00606 V=800.0 PL=0
MOVL C00607 V=800.0 PL=0
MOVL C00608 V=800.0 PL=0
MOVL C00609 V=800.0 PL=0
MOVL C00610 V=800.0 PL=0
MOVL C00611 V=800.0 PL=0
MOVL C00612 V=800.0 PL=0
MOVL C00613 V=800.0 PL=0
MOVL C00614 V=800.0 PL=0
MOVL C00615 V=800.0 PL=0
MOVL C00616 V=800.0 PL=0
MOVL C00617 V=800.0 PL=0
MOVL C00618 V=800.0 PL=0
MOVL C00619 V=800.0 PL=0
MOVL C00620 V=800.0 PL=0
MOVL C00621 V=800.0 PL=0
MOVL C00622 V=800.0 PL=0
MOVL C00623 V=800.0 PL=0
MOVL C00624 V=800.0 PL=0
MOVL C00625 V=800.0 PL=0
MOVL C00626 V=800.0 PL=0
MOVL C00627 V=800.0 PL=0
MOVL C00628 V=800.0 PL=0
MOVL C00629 V=800.0 PL=0
MOVL C00630 V=800.0 PL=0
MOVL C00631 V=800.0 PL=0
MOVL C00632 V=800.0 PL=0
MOVL C00633 V=800.0 PL=0
MOVL C00634 V=800.0 PL=0
MOVL C00635 V=800.0 PL=0
MOVL C00636 V=800.0 PL=0
MOVL C00637 V=800.0 PL=0
MOVL C00638 V=800.0 PL=0
MOVL C00639 V=800.0 PL=0
MOVL C00640 V=800.0 PL=0
MOVL C00641 V=800.0 PL=0
MOVL C00642 V=800.0 PL=0
MOVL C00643 V=800.0 PL=0
MOVL C00644 V=800.0 PL=0
MOVL C00645 V=800.0 PL=0
MOVL C00646 V=800.0 PL=0
MOVL C00647 V=800.0 PL=0
MOVL C00648 V=800.0 PL=0
MOVL C00649 V=800.0 PL=0
MOVL C00650 V=800.0 PL=0
MOVL C00651 V=800.0 PL=0
MOVL C00652 V=800.0 PL=0
MOVL C00653 V=800.0 PL=0
MOVL C00654 V=800.0 PL=0
MOVL C00655 V=800.0 PL=0
MOVL C00656 V=800.0 PL=0
MOVL C00657 V=800.0 PL=0
MOVL C00658 V=800.0 PL=0
MOVL C00659 V=800.0 PL=0
MOVL C00660 V=800.0 PL=0
MOVL C00661 V=800.0 PL=0
MOVL C00662 V=800.0 PL=0
MOVL C00663 V=800.0 PL=0
MOVL C00664 V=800.0 PL=0
MOVL C00665 V=800.0 PL=0
MOVL C00666 V=800.0 PL=0
MOVL C00667 V=800.0 PL=0
MOVL C00668 V=800.0 PL=0
MOVL C00669 V=800.0 PL=0
MOVL C00670 V=800.0 PL=0
MOVL C00671 V=800.0 PL=0
MOVL C00672 V=800.0 PL=0
MOVL C00673 V=800.0 PL=0
MOVL C00674 V=800.0 PL=0
MOVL C00675 V=800.0 PL=0
MOVL C00676 V=800.0 PL=0
MOVL C00677 V=800.0 PL=0
MOVL C00678 V=800.0 PL=0
MOVL C00679 V=800.0 PL=0
MOVL C00680 V=800.0 PL=0
MOVL C00681 V=800.0 PL=0
MOVL C00682 V=800.0 PL=0
MOVL C00683 V=800.0 PL=0
MOVL C00684 V=800.0 PL=0
MOVL C00685 V=800.0 PL=0
MOVL C00686 V=800.0 PL=0
MOVL C00687 V=800.0 PL=0
MOVL C00688 V=800.0 PL=0
MOVL C00689 V=800.0 PL=0
MOVL C00690 V=800.0 PL=0
MOVL C00691 V=800.0 PL=0
MOVL C00692 V=800.0 PL=0
MOVL C00693 V=800.0 PL=0
MOVL C00694 V=800.0 PL=0
MOVL C00695 V=800.0 PL=0
MOVL C00696 V=800.0 PL=0
MOVL C00697 V=800.0 PL=0
MOVL C00698 V=800.0 PL=0
MOVL C00699 V=800.0 PL=0
MOVL C00700 V=800.0 PL=0
MOVL C00701 V=800.0 PL=0
MOVL C00702 V=800.0 PL=0
MOVL C00703 V=800.0 PL=0
MOVL C00704 V=800.0 PL=0
MOVL C00705 V=800.0 PL=0
MOVL C00706 V=800.0 PL=0
MOVL C00707 V=800.0 PL=0
MOVL C00708 V=800.0 PL=0
MOVL C00709 V=800.0 PL=0
MOVL C00710 V=800.0 PL=0
MOVL C00711 V=800.0 PL=0
MOVL C00712 V=800.0 PL=0
MOVL C00713 V=800.0 PL=0
MOVL C00714 V=800.0 PL=0
MOVL C00715 V=800.0 PL=0
MOVL C00716 V=800.0 PL=0
MOVL C00717 V=800.0 PL=0
MOVL C00718 V=800.0 PL=0
MOVL C00719 V=800.0 PL=0
MOVL C00720 V=800.0 PL=0
MOVL C00721 V=800.0 PL=0
MOVL C00722 V=800.0 PL=0
MOVL C00723 V=800.0 PL=0
MOVL C00724 V=800.0 PL=0
MOVL C00725 V=800.0 PL=0
MOVL C00726 V=800.0 PL=0
MOVL C00727 V=800.0 PL=0
MOVL C00728 V=800.0 PL=0
MOVL C00729 V=800.0 PL=0
MOVL C00730 V=800.0 PL=0
MOVL C00731 V=800.0 PL=0
MOVL C00732 V=800.0 PL=0
MOVL C00733 V=800.0 PL=0
MOVL C00734 V=800.0 PL=0
MOVL C00735 V=800.0 PL=0
MOVL C00736 V=800.0 PL=0
MOVL C00737 V=800.0 PL=0
MOVL C00738 V=800.0 PL=0
MOVL C00739 V=800.0 PL=0
MOVL C00740 V=800.0 PL=0
MOVL C00741 V=800.0 PL=0
MOVL C00742 V=800.0 PL=0
MOVL C00743 V=800.0 PL=0
MOVL C00744 V=800.0 PL=0
MOVL C00745 V=800.0 PL=0
MOVL C00746 V=800.0 PL=0
MOVL C00747 V=800.0 PL=0
MOVL C00748 V=800.0 PL=0
MOVL C00749 V=800.0 PL=0
MOVL C00750 V=800.0 PL=0
MOVL C00751 V=800.0 PL=0
MOVL C00752 V=800.0 PL=0
MOVL C00753 V=800.0 PL=0
MOVL C00754 V=800.0 PL=0
MOVL C00755 V=800.0 PL=0
MOVL C00756 V=800.0 PL=0
MOVL C00757 V=800.0 PL=0
MOVL C00758 V=800.0 PL=0
MOVL C00759 V=800.0 PL=0
MOVL C00760 V=800.0 PL=0
MOVL C00761 V=800.0 PL=0
MOVL C00762 V=800.0 PL=0
MOVL C00763 V=800.0 PL=0
MOVL C00764 V=800.0 PL=0
MOVL C00765 V=800.0 PL=0
MOVL C00766 V=800.0 PL=0
MOVL C00767 V=800.0 PL=0
MOVL C00768 V=800.0 PL=0
MOVL C00769 V=800.0 PL=0
MOVL C00770 V=800.0 PL=0
MOVL C00771 V=800.0 PL=0
MOVL C00772 V=800.0 PL=0
MOVL C00773 V=800.0 PL=0
MOVL C00774 V=800.0 PL=0
MOVL C00775 V=800.0 PL=0
MOVL C00776 V=800.0 PL=0
MOVL C00777 V=800.0 PL=0
MOVL C00778 V=800.0 PL=0
MOVL C00779 V=800.0 PL=0
MOVL C00780 V=800.0 PL=0
MOVL C00781 V=800.0 PL=0
MOVL C00782 V=800.0 PL=0
MOVL C00783 V=800.0 PL=0
MOVL C00784 V=800.0 PL=0
MOVL C00785 V=800.0 PL=0
MOVL C00786 V=800.0 PL=0
MOVL C00787 V=800.0 PL=0
MOVL C00788 V=800.0 PL=0
MOVL C00789 V=800.0 PL=0
MOVL C00790 V=800.0 PL=0
MOVL C00791 V=800.0 PL=0
MOVL C00792 V=800.0 PL=0
MOVL C00793 V=800.0 PL=0
MOVL C00794 V=800.0 PL=0
MOVL C00795 V=800.0 PL=0
MOVL C00796 V=800.0 PL=0
MOVL C00797 V=800.0 PL=0
MOVL C00798 V=800.0 PL=0
MOVL C00799 V=800.0 PL=0
MOVL C00800 V=800.0 PL=0
MOVL C00801 V=800.0 PL=0
MOVL C00802 V=800.0 PL=0
MOVL C00803 V=800.0 PL=0
MOVL C00804 V=800.0 PL=0
MOVL C00805 V=800.0 PL=0
MOVL C00806 V=800.0 PL=0
MOVL C00807 V=800.0 PL=0
MOVL C00808 V=800.0 PL=0
MOVL C00809 V=800.0 PL=0
MOVL C00810 V=800.0 PL=0
MOVL C00811 V=800.0 PL=0
MOVL C00812 V=800.0 PL=0
MOVL C00813 V=800.0 PL=0
MOVL C00814 V=800.0 PL=0
MOVL C00815 V=800.0 PL=0
MOVL C00816 V=800.0 PL=0
MOVL C00817 V=800.0 PL=0
MOVL C00818 V=800.0 PL=0
MOVL C00819 V=800.0 PL=0
MOVL C00820 V=800.0 PL=0
MOVL C00821 V=800.0 PL=0
MOVL C00822 V=800.0 PL=0
MOVL C00823 V=800.0 PL=0
MOVL C00824 V=800.0 PL=0
MOVL C00825 V=800.0 PL=0
MOVL C00826 V=800.0 PL=0
MOVL C00827 V=800.0 PL=0
MOVL C00828 V=800.0 PL=0
MOVL C00829 V=800.0 PL=0
MOVL C00830 V=800.0 PL=0
MOVL C00831 V=800.0 PL=0
MOVL C00832 V=800.0 PL=0
MOVL C00833 V=800.0 PL=0
MOVL C00834 V=800.0 PL=0
MOVL C00835 V=800.0 PL=0
MOVL C00836 V=800.0 PL=0
MOVL C00837 V=800.0 PL=0
MOVL C00838 V=800.0 PL=0
MOVL C00839 V=800.0 PL=0
MOVL C00840 V=800.0 PL=0
MOVL C00841 V=800.0 PL=0
MOVL C00842 V=800.0 PL=0
MOVL C00843 V=800.0 PL=0
MOVL C00844 V=800.0 PL=0
MOVL C00845 V=800.0 PL=0
MOVL C00846 V=800.0 PL=0
MOVL C00847 V=800.0 PL=0
MOVL C00848 V=800.0 PL=0
MOVL C00849 V=800.0 PL=0
MOVL C00850 V=800.0 PL=0
MOVL C00851 V=800.0 PL=0
MOVL C00852 V=800.0 PL=0
MOVL C00853 V=800.0 PL=0
MOVL C00854 V=800.0 PL=0
MOVL C00855 V=800.0 PL=0
MOVL C00856 V=800.0 PL=0
MOVL C00857 V=800.0 PL=0
MOVL C00858 V=800.0 PL=0
MOVL C00859 V=800.0 PL=0
MOVL C00860 V=800.0 PL=0
MOVL C00861 V=800.0 PL=0
MOVL C00862 V=800.0 PL=0
MOVL C00863 V=800.0 PL=0
MOVL C00864 V=800.0 PL=0
MOVL C00865 V=800.0 PL=0
MOVL C00866 V=800.0 PL=0
MOVL C00867 V=800.0 PL=0
MOVL C00868 V=800.0 PL=0
MOVL C00869 V=800.0 PL=0
MOVL C00870 V=800.0 PL=0
MOVL C00871 V=800.0 PL=0
MOVL C00872 V=800.0 PL=0
MOVL C00873 V=800.0 PL=0
MOVL C00874 V=800.0 PL=0
MOVL C00875 V=800.0 PL=0
MOVL C00876 V=800.0 PL=0
MOVL C00877 V=800.0 PL=0
MOVL C00878 V=800.0 PL=0
MOVL C00879 V=800.0 PL=0
MOVL C00880 V=800.0 PL=0
MOVL C00881 V=800.0 PL=0
MOVL C00882 V=800.0 PL=0
MOVL C00883 V=800.0 PL=0
MOVL C00884 V=800.0 PL=0
MOVL C00885 V=800.0 PL=0
MOVL C00886 V=800.0 PL=0
MOVL C00887 V=800.0 PL=0
MOVL C00888 V=800.0 PL=0
MOVL C00889 V=800.0 PL=0
MOVL C00890 V=800.0 PL=0
MOVL C00891 V=800.0 PL=0
MOVL C00892 V=800.0 PL=0
MOVL C00893 V=800.0 PL=0
MOVL C00894 V=800.0 PL=0
MOVL C00895 V=800.0 PL=0
MOVL C00896 V=800.0 PL=0
MOVL C00897 V=800.0 PL=0
MOVL C00898 V=800.0 PL=0
MOVL C00899 V=800.0 PL=0
MOVL C00900 V=800.0 PL=0
MOVL C00901 V=800.0 PL=0
MOVL C00902 V=800.0 PL=0
MOVL C00903 V=800.0 PL=0
MOVL C00904 V=800.0 PL=0
MOVL C00905 V=800.0 PL=0
MOVL C00906 V=800.0 PL=0
MOVL C00907 V=800.0 PL=0
MOVL C00908 V=800.0 PL=0
MOVL C00909 V=800.0 PL=0
MOVL C00910 V=800.0 PL=0
MOVL C00911 V=800.0 PL=0
MOVL C00912 V=800.0 PL=0
MOVL C00913 V=800.0 PL=0
MOVL C00914 V=800.0 PL=0
MOVL C00915 V=800.0 PL=0
MOVL C00916 V=800.0 PL=0
MOVL C00917 V=800.0 PL=0
MOVL C00918 V=800.0 PL=0
MOVL C00919 V=800.0 PL=0
MOVL C00920 V=800.0 PL=0
MOVL C00921 V=800.0 PL=0
MOVL C00922 V=800.0 PL=0
MOVL C00923 V=800.0 PL=0
MOVL C00924 V=800.0 PL=0
MOVL C00925 V=800.0 PL=0
MOVL C00926 V=800.0 PL=0
MOVL C00927 V=800.0 PL=0
MOVL C00928 V=800.0 PL=0
MOVL C00929 V=800.0 PL=0
MOVL C00930 V=800.0 PL=0
MOVL C00931 V=800.0 PL=0
MOVL C00932 V=800.0 PL=0
MOVL C00933 V=800.0 PL=0
MOVL C00934 V=800.0 PL=0
MOVL C00935 V=800.0 PL=0
MOVL C00936 V=800.0 PL=0
MOVL C00937 V=800.0 PL=0
MOVL C00938 V=800.0 PL=0
MOVL C00939 V=800.0 PL=0
MOVL C00940 V=800.0 PL=0
MOVL C00941 V=800.0 PL=0
MOVL C00942 V=800.0 PL=0
MOVL C00943 V=800.0 PL=0
MOVL C00944 V=800.0 PL=0
MOVL C00945 V=800.0 PL=0
MOVL C00946 V=800.0 PL=0
MOVL C00947 V=800.0 PL=0
MOVL C00948 V=800.0 PL=0
MOVL C00949 V=800.0 PL=0
MOVL C00950 V=800.0 PL=0
MOVL C00951 V=800.0 PL=0
MOVL C00952 V=800.0 PL=0
MOVL C00953 V=800.0 PL=0
MOVL C00954 V=800.0 PL=0
MOVL C00955 V=800.0 PL=0
MOVL C00956 V=800.0 PL=0
MOVL C00957 V=800.0 PL=0
MOVL C00958 V=800.0 PL=0
MOVL C00959 V=800.0 PL=0
MOVL C00960 V=800.0 PL=0
MOVL C00961 V=800.0 PL=0
MOVL C00962 V=800.0 PL=0
MOVL C00963 V=800.0 PL=0
MOVL C00964 V=800.0 PL=0
MOVL C00965 V=800.0 PL=0
MOVL C00966 V=800.0 PL=0
MOVL C00967 V=800.0 PL=0
MOVL C00968 V=800.0 PL=0
MOVL C00969 V=800.0 PL=0
MOVL C00970 V=800.0 PL=0
MOVL C00971 V=800.0 PL=0
MOVL C00972 V=800.0 PL=0
MOVL C00973 V=800.0 PL=0
MOVL C00974 V=800.0 PL=0
MOVL C00975 V=800.0 PL=0
MOVL C00976 V=800.0 PL=0
MOVL C00977 V=800.0 PL=0
MOVL C00978 V=800.0 PL=0
MOVL C00979 V=800.0 PL=0
MOVL C00980 V=800.0 PL=0
MOVL C00981 V=800.0 PL=0
MOVL C00982 V=800.0 PL=0
MOVL C00983 V=800.0 PL=0
MOVL C00984 V=800.0 PL=0
MOVL C00985 V=800.0 PL=0
MOVL C00986 V=800.0 PL=0
MOVL C00987 V=800.0 PL=0
MOVL C00988 V=800.0 PL=0
MOVL C00989 V=800.0 PL=0
MOVL C00990 V=800.0 PL=0
MOVL C00991 V=800.0 PL=0
MOVL C00992 V=800.0 PL=0
MOVL C00993 V=800.0 PL=0
MOVL C00994 V=800.0 PL=0
MOVL C00995 V=800.0 PL=0
MOVL C00996 V=800.0 PL=0
MOVL C00997 V=800.0 PL=0
MOVL C00998 V=800.0 PL=0
MOVL C00999 V=800.0 PL=0
MOVL C01000 V=800.0 PL=0
MOVL C01001 V=800.0 PL=0
MOVL C01002 V=800.0 PL=0
MOVL C01003 V=800.0 PL=0
MOVL C01004 V=800.0 PL=0
MOVL C01005 V=800.0 PL=0
MOVL C01006 V=800.0 PL=0
MOVL C01007 V=800.0 PL=0
MOVL C01008 V=800.0 PL=0
MOVL C01009 V=800.0 PL=0
MOVL C01010 V=800.0 PL=0
MOVL C01011 V=800.0 PL=0
MOVL C01012 V=800.0 PL=0
MOVL C01013 V=800.0 PL=0
MOVL C01014 V=800.0 PL=0
MOVL C01015 V=800.0 PL=0
MOVL C01016 V=800.0 PL=0
MOVL C01017 V=800.0 PL=0
MOVL C01018 V=800.0 PL=0
MOVL C01019 V=800.0 PL=0
MOVL C01020 V=800.0 PL=0
MOVL C01021 V=800.0 PL=0
MOVL C01022 V=800.0 PL=0
MOVL C01023 V=800.0 PL=0
MOVL C01024 V=800.0 PL=0
MOVL C01025 V=800.0 PL=0
MOVL C01026 V=800.0 PL=0
MOVL C01027 V=800.0 PL=0
MOVL C01028 V=800.0 PL=0
MOVL C01029 V=800.0 PL=0
MOVL C01030 V=800.0 PL=0
MOVL C01031 V=800.0 PL=0
MOVL C01032 V=800.0 PL=0
MOVL C01033 V=800.0 PL=0
MOVL C01034 V=800.0 PL=0
MOVL C01035 V=800.0 PL=0
MOVL C01036 V=800.0 PL=0
MOVL C01037 V=800.0 PL=0
MOVL C01038 V=800.0 PL=0
MOVL C01039 V=800.0 PL=0
MOVL C01040 V=800.0 PL=0
MOVL C01041 V=800.0 PL=0
MOVL C01042 V=800.0 PL=0
MOVL C01043 V=800.0 PL=0
MOVL C01044 V=800.0 PL=0
MOVL C01045 V=800.0 PL=0
MOVL C01046 V=800.0 PL=0
MOVL C01047 V=800.0 PL=0
MOVL C01048 V=800.0 PL=0
MOVL C01049 V=800.0 PL=0
MOVL C01050 V=800.0 PL=0
MOVL C01051 V=800.0 PL=0
MOVL C01052 V=800.0 PL=0
MOVL C01053 V=800.0 PL=0
MOVL C01054 V=800.0 PL=0
MOVL C01055 V=800.0 PL=0
MOVL C01056 V=800.0 PL=0
MOVL C01057 V=800.0 PL=0
MOVL C01058 V=800.0 PL=0
MOVL C01059 V=800.0 PL=0
MOVL C01060 V=800.0 PL=0
MOVL C01061 V=800.0 PL=0
MOVL C01062 V=800.0 PL=0
MOVL C01063 V=800.0 PL=0
MOVL C01064 V=800.0 PL=0
MOVL C01065 V=800.0 PL=0
MOVL C01066 V=800.0 PL=0
MOVL C01067 V=800.0 PL=0
MOVL C01068 V=800.0 PL=0
MOVL C01069 V=800.0 PL=0
MOVL C01070 V=800.0 PL=0
MOVL C01071 V=800.0 PL=0
MOVL C01072 V=800.0 PL=0
MOVL C01073 V=800.0 PL=0
MOVL C01074 V=800.0 PL=0
MOVL C01075 V=800.0 PL=0
MOVL C01076 V=800.0 PL=0
MOVL C01077 V=800.0 PL=0
MOVL C01078 V=800.0 PL=0
MOVL C01079 V=800.0 PL=0
MOVL C01080 V=800.0 PL=0
MOVL C01081 V=800.0 PL=0
MOVL C01082 V=800.0 PL=0
MOVL C01083 V=800.0 PL=0
MOVL C01084 V=800.0 PL=0
MOVL C01085 V=800.0 PL=0
MOVL C01086 V=800.0 PL=0
MOVL C01087 V=800.0 PL=0
MOVL C01088 V=800.0 PL=0
MOVL C01089 V=800.0 PL=0
MOVL C01090 V=800.0 PL=0
MOVL C01091 V=800.0 PL=0
MOVL C01092 V=800.0 PL=0
MOVL C01093 V=800.0 PL=0
MOVL C01094 V=800.0 PL=0
MOVL C01095 V=800.0 PL=0
MOVL C01096 V=800.0 PL=0
MOVL C01097 V=800.0 PL=0
MOVL C01098 V=800.0 PL=0
MOVL C01099 V=800.0 PL=0
MOVL C01100 V=800.0 PL=0
MOVL C01101 V=800.0 PL=0
MOVL C01102 V=800.0 PL=0
MOVL C01103 V=800.0 PL=0
MOVL C01104 V=800.0 PL=0
MOVL C01105 V=800.0 PL=0
MOVL C01106 V=800.0 PL=0
MOVL C01107 V=800.0 PL=0
MOVL C01108 V=800.0 PL=0
MOVL C01109 V=800.0 PL=0
MOVL C01110 V=800.0 PL=0
MOVL C01111 V=800.0 PL=0
MOVL C01112 V=800.0 PL=0
MOVL C01113 V=800.0 PL=0
MOVL C01114 V=800.0 PL=0
MOVL C01115 V=800.0 PL=0
MOVL C01116 V=800.0 PL=0
MOVL C01117 V=800.0 PL=0
MOVL C01118 V=800.0 PL=0
MOVL C01119 V=800.0 PL=0
MOVL C01120 V=800.0 PL=0
MOVL C01121 V=800.0 PL=0
MOVL C01122 V=800.0 PL=0
MOVL C01123 V=800.0 PL=0
MOVL C01124 V=800.0 PL=0
MOVL C01125 V=800.0 PL=0
MOVL C01126 V=800.0 PL=0
MOVL C01127 V=800.0 PL=0
MOVL C01128 V=800.0 PL=0
MOVL C01129 V=800.0 PL=0
MOVL C01130 V=800.0 PL=0
MOVL C01131 V=800.0 PL=0
MOVL C01132 V=800.0 PL=0
MOVL C01133 V=800.0 PL=0
MOVL C01134 V=800.0 PL=0
MOVL C01135 V=800.0 PL=0
MOVL C01136 V=800.0 PL=0
MOVL C01137 V=800.0 PL=0
MOVL C01138 V=800.0 PL=0
MOVL C01139 V=800.0 PL=0
MOVL C01140 V=800.0 PL=0
MOVL C01141 V=800.0 PL=0
MOVL C01142 V=800.0 PL=0
MOVL C01143 V=800.0 PL=0
MOVL C01144 V=800.0 PL=0
MOVL C01145 V=800.0 PL=0
MOVL C01146 V=800.0 PL=0
MOVL C01147 V=800.0 PL=0
MOVL C01148 V=800.0 PL=0
MOVL C01149 V=800.0 PL=0
MOVL C01150 V=800.0 PL=0
MOVL C01151 V=800.0 PL=0
MOVL C01152 V=800.0 PL=0
MOVL C01153 V=800.0 PL=0
MOVL C01154 V=800.0 PL=0
MOVL C01155 V=800.0 PL=0
MOVL C01156 V=800.0 PL=0
MOVL C01157 V=800.0 PL=0
MOVL C01158 V=800.0 PL=0
MOVL C01159 V=800.0 PL=0
MOVL C01160 V=800.0 PL=0
MOVL C01161 V=800.0 PL=0
MOVL C01162 V=800.0 PL=0
MOVL C01163 V=800.0 PL=0
MOVL C01164 V=800.0 PL=0
MOVL C01165 V=800.0 PL=0
MOVL C01166 V=800.0 PL=0
MOVL C01167 V=800.0 PL=0
MOVL C01168 V=800.0 PL=0
MOVL C01169 V=800.0 PL=0
MOVL C01170 V=800.0 PL=0
MOVL C01171 V=800.0 PL=0
MOVL C01172 V=800.0 PL=0
MOVL C01173 V=800.0 PL=0
MOVL C01174 V=800.0 PL=0
MOVL C01175 V=800.0 PL=0
MOVL C01176 V=800.0 PL=0
MOVL C01177 V=800.0 PL=0
MOVL C01178 V=800.0 PL=0
MOVL C01179 V=800.0 PL=0
MOVL C01180 V=800.0 PL=0
MOVL C01181 V=800.0 PL=0
MOVL C01182 V=800.0 PL=0
MOVL C01183 V=800.0 PL=0
MOVL C01184 V=800.0 PL=0
MOVL C01185 V=800.0 PL=0
MOVL C01186 V=800.0 PL=0
MOVL C01187 V=800.0 PL=0
MOVL C01188 V=800.0 PL=0
MOVL C01189 V=800.0 PL=0
MOVL C01190 V=800.0 PL=0
MOVL C01191 V=800.0 PL=0
MOVL C01192 V=800.0 PL=0
MOVL C01193 V=800.0 PL=0
MOVL C01194 V=800.0 PL=0
MOVL C01195 V=800.0 PL=0
MOVL C01196 V=800.0 PL=0
MOVL C01197 V=800.0 PL=0
MOVL C01198 V=800.0 PL=0
MOVL C01199 V=800.0 PL=0
MOVL C01200 V=800.0 PL=0
MOVL C01201 V=800.0 PL=0
MOVL C01202 V=800.0 PL=0
MOVL C01203 V=800.0 PL=0
MOVL C01204 V=800.0 PL=0
MOVL C01205 V=800.0 PL=0
MOVL C01206 V=800.0 PL=0
MOVL C01207 V=800.0 PL=0
MOVL C01208 V=800.0 PL=0
MOVL C01209 V=800.0 PL=0
MOVL C01210 V=800.0 PL=0
MOVL C01211 V=800.0 PL=0
MOVL C01212 V=800.0 PL=0
MOVL C01213 V=800.0 PL=0
MOVL C01214 V=800.0 PL=0
MOVL C01215 V=800.0 PL=0
MOVL C01216 V=800.0 PL=0
MOVL C01217 V=800.0 PL=0
MOVL C01218 V=800.0 PL=0
MOVL C01219 V=800.0 PL=0
MOVL C01220 V=800.0 PL=0
MOVL C01221 V=800.0 PL=0
MOVL C01222 V=800.0 PL=0
MOVL C01223 V=800.0 PL=0
MOVL C01224 V=800.0 PL=0
MOVL C01225 V=800.0 PL=0
MOVL C01226 V=800.0 PL=0
MOVL C01227 V=800.0 PL=0
MOVL C01228 V=800.0 PL=0
MOVL C01229 V=800.0 PL=0
MOVL C01230 V=800.0 PL=0
MOVL C01231 V=800.0 PL=0
MOVL C01232 V=800.0 PL=0
MOVL C01233 V=800.0 PL=0
MOVL C01234 V=800.0 PL=0
MOVL C01235 V=800.0 PL=0
MOVL C01236 V=800.0 PL=0
MOVL C01237 V=800.0 PL=0
MOVL C01238 V=800.0 PL=0
MOVL C01239 V=800.0 PL=0
MOVL C01240 V=800.0 PL=0
MOVL C01241 V=800.0 PL=0
MOVL C01242 V=800.0 PL=0
MOVL C01243 V=800.0 PL=0
MOVL C01244 V=800.0 PL=0
MOVL C01245 V=800.0 PL=0
MOVL C01246 V=800.0 PL=0
MOVL C01247 V=800.0 PL=0
MOVL C01248 V=800.0 PL=0
MOVL C01249 V=800.0 PL=0
MOVL C01250 V=800.0 PL=0
MOVL C01251 V=800.0 PL=0
MOVL C01252 V=800.0 PL=0
MOVL C01253 V=800.0 PL=0
MOVL C01254 V=800.0 PL=0
MOVL C01255 V=800.0 PL=0
MOVL C01256 V=800.0 PL=0
MOVL C01257 V=800.0 PL=0
MOVL C01258 V=800.0 PL=0
MOVL C01259 V=800.0 PL=0
MOVL C01260 V=800.0 PL=0
MOVL C01261 V=800.0 PL=0
MOVL C01262 V=800.0 PL=0
MOVL C01263 V=800.0 PL=0
MOVL C01264 V=800.0 PL=0
MOVL C01265 V=800.0 PL=0
MOVL C01266 V=800.0 PL=0
MOVL C01267 V=800.0 PL=0
MOVL C01268 V=800.0 PL=0
MOVL C01269 V=800.0 PL=0
MOVL C01270 V=800.0 PL=0
MOVL C01271 V=800.0 PL=0
MOVL C01272 V=800.0 PL=0
MOVL C01273 V=800.0 PL=0
MOVL C01274 V=800.0 PL=0
MOVL C01275 V=800.0 PL=0
MOVL C01276 V=800.0 PL=0
MOVL C01277 V=800.0 PL=0
MOVL C01278 V=800.0 PL=0
MOVL C01279 V=800.0 PL=0
MOVL C01280 V=800.0 PL=0
MOVL C01281 V=800.0 PL=0
MOVL C01282 V=800.0 PL=0
MOVL C01283 V=800.0 PL=0
MOVL C01284 V=800.0 PL=0
MOVL C01285 V=800.0 PL=0
MOVL C01286 V=800.0 PL=0
MOVL C01287 V=800.0 PL=0
MOVL C01288 V=800.0 PL=0
MOVL C01289 V=800.0 PL=0
MOVL C01290 V=800.0 PL=0
MOVL C01291 V=800.0 PL=0
MOVL C01292 V=800.0 PL=0
MOVL C01293 V=800.0 PL=0
MOVL C01294 V=800.0 PL=0
MOVL C01295 V=800.0 PL=0
MOVL C01296 V=800.0 PL=0
MOVL C01297 V=800.0 PL=0
MOVL C01298 V=800.0 PL=0
MOVL C01299 V=800.0 PL=0
MOVL C01300 V=800.0 PL=0
MOVL C01301 V=800.0 PL=0
MOVL C01302 V=800.0 PL=0
MOVL C01303 V=800.0 PL=0
MOVL C01304 V=800.0 PL=0
MOVL C01305 V=800.0 PL=0
MOVL C01306 V=800.0 PL=0
MOVL C01307 V=800.0 PL=0
MOVL C01308 V=800.0 PL=0
MOVL C01309 V=800.0 PL=0
MOVL C01310 V=800.0 PL=0
MOVL C01311 V=800.0 PL=0
MOVL C01312 V=800.0 PL=0
MOVL C01313 V=800.0 PL=0
MOVL C01314 V=800.0 PL=0
MOVL C01315 V=800.0 PL=0
MOVL C01316 V=800.0 PL=0
MOVL C01317 V=800.0 PL=0
MOVL C01318 V=800.0 PL=0
MOVL C01319 V=800.0 PL=0
MOVL C01320 V=800.0 PL=0
MOVL C01321 V=800.0 PL=0
MOVL C01322 V=800.0 PL=0
MOVL C01323 V=800.0 PL=0
MOVL C01324 V=800.0 PL=0
MOVL C01325 V=800.0 PL=0
MOVL C01326 V=800.0 PL=0
MOVL C01327 V=800.0 PL=0
MOVL C01328 V=800.0 PL=0
MOVL C01329 V=800.0 PL=0
MOVL C01330 V=800.0 PL=0
MOVL C01331 V=800.0 PL=0
MOVL C01332 V=800.0 PL=0
MOVL C01333 V=800.0 PL=0
MOVL C01334 V=800.0 PL=0
MOVL C01335 V=800.0 PL=0
MOVL C01336 V=800.0 PL=0
MOVL C01337 V=800.0 PL=0
MOVL C01338 V=800.0 PL=0
MOVL C01339 V=800.0 PL=0
MOVL C01340 V=800.0 PL=0
MOVL C01341 V=800.0 PL=0
MOVL C01342 V=800.0 PL=0
MOVL C01343 V=800.0 PL=0
MOVL C01344 V=800.0 PL=0
MOVL C01345 V=800.0 PL=0
MOVL C01346 V=800.0 PL=0
MOVL C01347 V=800.0 PL=0
MOVL C01348 V=800.0 PL=0
MOVL C01349 V=800.0 PL=0
MOVL C01350 V=800.0 PL=0
MOVL C01351 V=800.0 PL=0
MOVL C01352 V=800.0 PL=0
MOVL C01353 V=800.0 PL=0
MOVL C01354 V=800.0 PL=0
MOVL C01355 V=800.0 PL=0
MOVL C01356 V=800.0 PL=0
MOVL C01357 V=800.0 PL=0
MOVL C01358 V=800.0 PL=0
MOVL C01359 V=800.0 PL=0
MOVL C01360 V=800.0 PL=0
MOVL C01361 V=800.0 PL=0
MOVL C01362 V=800.0 PL=0
MOVL C01363 V=800.0 PL=0
MOVL C01364 V=800.0 PL=0
MOVL C01365 V=800.0 PL=0
MOVL C01366 V=800.0 PL=0
MOVL C01367 V=800.0 PL=0
MOVL C01368 V=800.0 PL=0
MOVL C01369 V=800.0 PL=0
MOVL C01370 V=800.0 PL=0
MOVL C01371 V=800.0 PL=0
MOVL C01372 V=800.0 PL=0
MOVL C01373 V=800.0 PL=0
MOVL C01374 V=800.0 PL=0
MOVL C01375 V=800.0 PL=0
MOVL C01376 V=800.0 PL=0
MOVL C01377 V=800.0 PL=0
MOVL C01378 V=800.0 PL=0
MOVL C01379 V=800.0 PL=0
MOVL C01380 V=800.0 PL=0
MOVL C01381 V=800.0 PL=0
MOVL C01382 V=800.0 PL=0
MOVL C01383 V=800.0 PL=0
MOVL C01384 V=800.0 PL=0
MOVL C01385 V=800.0 PL=0
MOVL C01386 V=800.0 PL=0
MOVL C01387 V=800.0 PL=0
MOVL C01388 V=800.0 PL=0
MOVL C01389 V=800.0 PL=0
MOVL C01390 V=800.0 PL=0
MOVL C01391 V=800.0 PL=0
MOVL C01392 V=800.0 PL=0
MOVL C01393 V=800.0 PL=0
MOVL C01394 V=800.0 PL=0
MOVL C01395 V=800.0 PL=0
MOVL C01396 V=800.0 PL=0
MOVL C01397 V=800.0 PL=0
MOVL C01398 V=800.0 PL=0
MOVL C01399 V=800.0 PL=0
MOVL C01400 V=800.0 PL=0
MOVL C01401 V=800.0 PL=0
MOVL C01402 V=800.0 PL=0
MOVL C01403 V=800.0 PL=0
MOVL C01404 V=800.0 PL=0
MOVL C01405 V=800.0 PL=0
MOVL C01406 V=800.0 PL=0
MOVL C01407 V=800.0 PL=0
MOVL C01408 V=800.0 PL=0
MOVL C01409 V=800.0 PL=0
MOVL C01410 V=800.0 PL=0
MOVL C01411 V=800.0 PL=0
MOVL C01412 V=800.0 PL=0
MOVL C01413 V=800.0 PL=0
MOVL C01414 V=800.0 PL=0
MOVL C01415 V=800.0 PL=0
MOVL C01416 V=800.0 PL=0
MOVL C01417 V=800.0 PL=0
MOVL C01418 V=800.0 PL=0
MOVL C01419 V=800.0 PL=0
MOVL C01420 V=800.0 PL=0
MOVL C01421 V=800.0 PL=0
MOVL C01422 V=800.0 PL=0
MOVL C01423 V=800.0 PL=0
MOVL C01424 V=800.0 PL=0
MOVL C01425 V=800.0 PL=0
MOVL C01426 V=800.0 PL=0
MOVL C01427 V=800.0 PL=0
MOVL C01428 V=800.0 PL=0
MOVL C01429 V=800.0 PL=0
MOVL C01430 V=800.0 PL=0
MOVL C01431 V=800.0 PL=0
MOVL C01432 V=800.0 PL=0
MOVL C01433 V=800.0 PL=0
MOVL C01434 V=800.0 PL=0
MOVL C01435 V=800.0 PL=0
MOVL C01436 V=800.0 PL=0
MOVL C01437 V=800.0 PL=0
MOVL C01438 V=800.0 PL=0
MOVL C01439 V=800.0 PL=0
MOVL C01440 V=800.0 PL=0
MOVL C01441 V=800.0 PL=0
MOVL C01442 V=800.0 PL=0
MOVL C01443 V=800.0 PL=0
MOVL C01444 V=800.0 PL=0
MOVL C01445 V=800.0 PL=0
MOVL C01446 V=800.0 PL=0
MOVL C01447 V=800.0 PL=0
MOVL C01448 V=800.0 PL=0
MOVL C01449 V=800.0 PL=0
MOVL C01450 V=800.0 PL=0
MOVL C01451 V=800.0 PL=0
MOVL C01452 V=800.0 PL=0
MOVL C01453 V=800.0 PL=0
MOVL C01454 V=800.0 PL=0
MOVL C01455 V=800.0 PL=0
MOVL C01456 V=800.0 PL=0
MOVL C01457 V=800.0 PL=0
MOVL C01458 V=800.0 PL=0
MOVL C01459 V=800.0 PL=0
MOVL C01460 V=800.0 PL=0
MOVL C01461 V=800.0 PL=0
MOVL C01462 V=800.0 PL=0
MOVL C01463 V=800.0 PL=0
MOVL C01464 V=800.0 PL=0
MOVL C01465 V=800.0 PL=0
MOVL C01466 V=800.0 PL=0
MOVL C01467 V=800.0 PL=0
MOVL C01468 V=800.0 PL=0
MOVL C01469 V=800.0 PL=0
MOVL C01470 V=800.0 PL=0
MOVL C01471 V=800.0 PL=0
MOVL C01472 V=800.0 PL=0
MOVL C01473 V=800.0 PL=0
MOVL C01474 V=800.0 PL=0
MOVL C01475 V=800.0 PL=0
MOVL C01476 V=800.0 PL=0
MOVL C01477 V=800.0 PL=0
MOVL C01478 V=800.0 PL=0
MOVL C01479 V=800.0 PL=0
MOVL C01480 V=800.0 PL=0
MOVL C01481 V=800.0 PL=0
MOVL C01482 V=800.0 PL=0
MOVL C01483 V=800.0 PL=0
MOVL C01484 V=800.0 PL=0
MOVL C01485 V=800.0 PL=0
MOVL C01486 V=800.0 PL=0
MOVL C01487 V=800.0 PL=0
MOVL C01488 V=800.0 PL=0
MOVL C01489 V=800.0 PL=0
MOVL C01490 V=800.0 PL=0
MOVL C01491 V=800.0 PL=0
MOVL C01492 V=800.0 PL=0
MOVL C01493 V=800.0 PL=0
MOVL C01494 V=800.0 PL=0
MOVL C01495 V=800.0 PL=0
MOVL C01496 V=800.0 PL=0
MOVL C01497 V=800.0 PL=0
MOVL C01498 V=800.0 PL=0
MOVL C01499 V=800.0 PL=0
MOVL C01500 V=800.0 PL=0
MOVL C01501 V=800.0 PL=0
MOVL C01502 V=800.0 PL=0
MOVL C01503 V=800.0 PL=0
MOVL C01504 V=800.0 PL=0
MOVL C01505 V=800.0 PL=0
MOVL C01506 V=800.0 PL=0
MOVL C01507 V=800.0 PL=0
MOVL C01508 V=800.0 PL=0
MOVL C01509 V=800.0 PL=0
MOVL C01510 V=800.0 PL=0
MOVL C01511 V=800.0 PL=0
MOVL C01512 V=800.0 PL=0
MOVL C01513 V=800.0 PL=0
MOVL C01514 V=800.0 PL=0
MOVL C01515 V=800.0 PL=0
MOVL C01516 V=800.0 PL=0
MOVL C01517 V=800.0 PL=0
MOVL C01518 V=800.0 PL=0
MOVL C01519 V=800.0 PL=0
MOVL C01520 V=800.0 PL=0
MOVL C01521 V=800.0 PL=0
MOVL C01522 V=800.0 PL=0
MOVL C01523 V=800.0 PL=0
MOVL C01524 V=800.0 PL=0
MOVL C01525 V=800.0 PL=0
MOVL C01526 V=800.0 PL=0
MOVL C01527 V=800.0 PL=0
MOVL C01528 V=800.0 PL=0
MOVL C01529 V=800.0 PL=0
MOVL C01530 V=800.0 PL=0
MOVL C01531 V=800.0 PL=0
MOVL C01532 V=800.0 PL=0
MOVL C01533 V=800.0 PL=0
MOVL C01534 V=800.0 PL=0
MOVL C01535 V=800.0 PL=0
MOVL C01536 V=800.0 PL=0
MOVL C01537 V=800.0 PL=0
MOVL C01538 V=800.0 PL=0
MOVL C01539 V=800.0 PL=0
MOVL C01540 V=800.0 PL=0
MOVL C01541 V=800.0 PL=0
MOVL C01542 V=800.0 PL=0
MOVL C01543 V=800.0 PL=0
MOVL C01544 V=800.0 PL=0
MOVL C01545 V=800.0 PL=0
MOVL C01546 V=800.0 PL=0
MOVL C01547 V=800.0 PL=0
MOVL C01548 V=800.0 PL=0
MOVL C01549 V=800.0 PL=0
MOVL C01550 V=800.0 PL=0
MOVL C01551 V=800.0 PL=0
MOVL C01552 V=800.0 PL=0
MOVL C01553 V=800.0 PL=0
MOVL C01554 V=800.0 PL=0
MOVL C01555 V=800.0 PL=0
MOVL C01556 V=800.0 PL=0
MOVL C01557 V=800.0 PL=0
MOVL C01558 V=800.0 PL=0
MOVL C01559 V=800.0 PL=0
MOVL C01560 V=800.0 PL=0
MOVL C01561 V=800.0 PL=0
MOVL C01562 V=800.0 PL=0
MOVL C01563 V=800.0 PL=0
MOVL C01564 V=800.0 PL=0
MOVL C01565 V=800.0 PL=0
MOVL C01566 V=800.0 PL=0
MOVL C01567 V=800.0 PL=0
MOVL C01568 V=800.0 PL=0
MOVL C01569 V=800.0 PL=0
MOVL C01570 V=800.0 PL=0
MOVL C01571 V=800.0 PL=0
MOVL C01572 V=800.0 PL=0
MOVL C01573 V=800.0 PL=0
MOVL C01574 V=800.0 PL=0
MOVL C01575 V=800.0 PL=0
MOVL C01576 V=800.0 PL=0
MOVL C01577 V=800.0 PL=0
MOVL C01578 V=800.0 PL=0
MOVL C01579 V=800.0 PL=0
MOVL C01580 V=800.0 PL=0
MOVL C01581 V=800.0 PL=0
MOVL C01582 V=800.0 PL=0
MOVL C01583 V=800.0 PL=0
MOVL C01584 V=800.0 PL=0
MOVL C01585 V=800.0 PL=0
MOVL C01586 V=800.0 PL=0
MOVL C01587 V=800.0 PL=0
MOVL C01588 V=800.0 PL=0
MOVL C01589 V=800.0 PL=0
MOVL C01590 V=800.0 PL=0
MOVL C01591 V=800.0 PL=0
MOVL C01592 V=800.0 PL=0
MOVL C01593 V=800.0 PL=0
MOVL C01594 V=800.0 PL=0
MOVL C01595 V=800.0 PL=0
MOVL C01596 V=800.0 PL=0
MOVL C01597 V=800.0 PL=0
MOVL C01598 V=800.0 PL=0
MOVL C01599 V=800.0 PL=0
MOVL C01600 V=800.0 PL=0
MOVL C01601 V=800.0 PL=0
MOVL C01602 V=800.0 PL=0
MOVL C01603 V=800.0 PL=0
MOVL C01604 V=800.0 PL=0
MOVL C01605 V=800.0 PL=0
MOVL C01606 V=800.0 PL=0
MOVL C01607 V=800.0 PL=0
MOVL C01608 V=800.0 PL=0
MOVL C01609 V=800.0 PL=0
MOVL C01610 V=800.0 PL=0
MOVL C01611 V=800.0 PL=0
MOVL C01612 V=800.0 PL=0
MOVL C01613 V=800.0 PL=0
MOVL C01614 V=800.0 PL=0
MOVL C01615 V=800.0 PL=0
MOVL C01616 V=800.0 PL=0
MOVL C01617 V=800.0 PL=0
MOVL C01618 V=800.0 PL=0
MOVL C01619 V=800.0 PL=0
MOVL C01620 V=800.0 PL=0
MOVL C01621 V=800.0 PL=0
MOVL C01622 V=800.0 PL=0
MOVL C01623 V=800.0 PL=0
MOVL C01624 V=800.0 PL=0
MOVL C01625 V=800.0 PL=0
MOVL C01626 V=800.0 PL=0
MOVL C01627 V=800.0 PL=0
MOVL C01628 V=800.0 PL=0
MOVL C01629 V=800.0 PL=0
MOVL C01630 V=800.0 PL=0
MOVL C01631 V=800.0 PL=0
MOVL C01632 V=800.0 PL=0
MOVL C01633 V=800.0 PL=0
MOVL C01634 V=800.0 PL=0
MOVL C01635 V=800.0 PL=0
MOVL C01636 V=800.0 PL=0
MOVL C01637 V=800.0 PL=0
MOVL C01638 V=800.0 PL=0
MOVL C01639 V=800.0 PL=0
MOVL C01640 V=800.0 PL=0
MOVL C01641 V=800.0 PL=0
MOVL C01642 V=800.0 PL=0
MOVL C01643 V=800.0 PL=0
MOVL C01644 V=800.0 PL=0
MOVL C01645 V=800.0 PL=0
MOVL C01646 V=800.0 PL=0
MOVL C01647 V=800.0 PL=0
MOVL C01648 V=800.0 PL=0
MOVL C01649 V=800.0 PL=0
MOVL C01650 V=800.0 PL=0
MOVL C01651 V=800.0 PL=0
MOVL C01652 V=800.0 PL=0
MOVL C01653 V=800.0 PL=0
MOVL C01654 V=800.0 PL=0
MOVL C01655 V=800.0 PL=0
MOVL C01656 V=800.0 PL=0
MOVL C01657 V=800.0 PL=0
MOVL C01658 V=800.0 PL=0
MOVL C01659 V=800.0 PL=0
